(* CoDeSys 2.3 project: test.pro *)
(* Title: cy-wg-06 - ClevergyAS *)
(* Author: Andrea Ravasio *)
(* Libraries: Standard.lib 8.11.10 12:37:48, Util.lib 26.9.14 11:12:46, mod_com.lib 8.11.10 12:37:48, SerComm.lib 31.5.11 09:06:48, Serial_Interface_01.lib 22.4.13 12:50:14, 32_Bit\Modb_l05.lib 8.8.11 17:34:10, WagoLibIdent.lib 25.2.13 13:49:34, WagoLibStatus.lib 8.11.10 12:37:48, SysLibFile.lib 8.11.10 12:37:48, SysLibRtc.lib 8.11.10 12:37:48, SysLibSockets.lib 5.5.11 09:22:24, SysLibEvent.lib 8.11.10 12:37:48, SysLibPlcCtrl.lib 8.11.10 12:37:48, SysLibCallback.lib 8.11.10 12:37:48, Ethernet.lib 8.11.10 12:37:48, WagoLibModbus_IP_01.lib 26.5.15 11:20:08, WagoLibMBX_01.lib 20.3.12 16:32:38, LON_01.lib 28.9.12 14:05:10 *)

(* PLC configuration (modules and I/O channels)
0750-1506 8DI / 8DO 24V DC 0.5A [Type_34_8_Channels] node 0, in %IB32 out %QB8 {INTTypePAAssignment = PLC; INTTypeModule = plugged}
  VPN_ST1 AT %IX16.0 [BOOLOnX_I] Ch_1 Digital input
  LAMP_AL AT %QX4.0 [BOOLOnX_Q] Ch_1 Digital output
  KEY_QE_ST AT %IX16.1 [BOOLOnX_I] Ch_2 Digital input
  CIR05_EN AT %QX4.1 [BOOLOnX_Q] Ch_2 Digital output
  CIR06_AL AT %IX16.2 [BOOLOnX_I] Ch_3 Digital input
  CIR03_EN AT %QX4.2 [BOOLOnX_Q] Ch_3 Digital output
  CIR06_ST AT %IX16.3 [BOOLOnX_I] Ch_4 Digital input
  CIR04_EN AT %QX4.3 [BOOLOnX_Q] Ch_4 Digital output
  CIR06_AUT AT %IX16.4 [BOOLOnX_I] Ch_5 Digital input
  CIR02_EN AT %QX4.4 [BOOLOnX_Q] Ch_5 Digital output
  CIR05_AL AT %IX16.5 [BOOLOnX_I] Ch_6 Digital input
  CIR01_EN AT %QX4.5 [BOOLOnX_Q] Ch_6 Digital output
  CIR05_ST AT %IX16.6 [BOOLOnX_I] Ch_7 Digital input
  CAL01_Rst_Bruc AT %QX4.6 [BOOLOnX_Q] Ch_7 Digital output
  CIR05_AUT AT %IX16.7 [BOOLOnX_I] Ch_8 Digital input
  CAL01_On_Off AT %QX4.7 [BOOLOnX_Q] Ch_8 Digital output
0750-0430 8 DI 24 V DC 3.0ms [Type_1_8_Channels] node 1, in %IB32 out %QB8 {INTTypePAAssignment = PLC; INTTypeModule = plugged}
  CIR02_ST AT %IX16.8 [BOOLOnX_I] Ch_1 Digital input
  CIR01_AUT AT %IX16.9 [BOOLOnX_I] Ch_2 Digital input
  CIR03_AL AT %IX16.10 [BOOLOnX_I] Ch_3 Digital input
  CIR04_ST AT %IX16.11 [BOOLOnX_I] Ch_4 Digital input
  CIR04_AL AT %IX16.12 [BOOLOnX_I] Ch_5 Digital input
  CIR02_AL AT %IX16.13 [BOOLOnX_I] Ch_6 Digital input
  CIR01_ST AT %IX16.14 [BOOLOnX_I] Ch_7 Digital input
  CAL01_ST AT %IX16.15 [BOOLOnX_I] Ch_8 Digital input
0750-0430 8 DI 24 V DC 3.0ms [Type_1_8_Channels] node 2, in %IB33 out %QB9 {INTTypePAAssignment = PLC; INTTypeModule = plugged}
  CAL01_AL AT %IX17.0 [BOOLOnX_I] Ch_1 Digital input
  CIR03_AUT AT %IX17.1 [BOOLOnX_I] Ch_2 Digital input
  CTL01_ST AT %IX17.2 [BOOLOnX_I] Ch_3 Digital input
  CIR01_AL AT %IX17.3 [BOOLOnX_I] Ch_4 Digital input
  CIR02_AUT AT %IX17.4 [BOOLOnX_I] Ch_5 Digital input
  ALARM_PM_PB_TB AT %IX17.5 [BOOLOnX_I] Ch_6 Digital input
  CIR03_ST AT %IX17.6 [BOOLOnX_I] Ch_7 Digital input
  CIR04_AUT AT %IX17.7 [BOOLOnX_I] Ch_8 Digital input
0750-0504 4 DO 24V DC 0.5A [Type_10_4_Channels] node 3, in %IB34 out %QB9 {INTTypePAAssignment = PLC; INTTypeModule = plugged}
  CIR06_EN AT %QX4.8 [BOOLOnX_Q] Ch_1 Digital output
  AT %QX4.9 [BOOLOnX_Q] Ch_2 Digital output
  AT %QX4.10 [BOOLOnX_Q] Ch_3 Digital output
  AT %QX4.11 [BOOLOnX_Q] Ch_4 Digital output
0750-0464#04 2/4 AI RTD / ADJ./ HA [Type_44_4_Channels] node 5, in %IB32 out %QB4 {INTTypePAAssignment = PLC; INTTypeModule = plugged}
  AT %IW0 [INTOnW_I] Ch_1 signed Input value
  AT %IW1 [INTOnW_I] Ch_2 signed Input value
  AT %IW2 [INTOnW_I] Ch_3 signed Input value
  T_S04 AT %IW3 [INTOnW_I] Ch_4 signed Input value
0750-0464#04 2/4 AI RTD / ADJ./ HA [Type_44_4_Channels] node 6, in %IB32 out %QB4 {INTTypePAAssignment = PLC; INTTypeModule = plugged}
  T_S05 AT %IW4 [INTOnW_I] Ch_1 signed Input value
  T_S08 AT %IW5 [INTOnW_I] Ch_2 signed Input value
  T_S06 AT %IW6 [INTOnW_I] Ch_3 signed Input value
  T_S09 AT %IW7 [INTOnW_I] Ch_4 signed Input value
0750-0464#04 2/4 AI RTD / ADJ./ HA [Type_44_4_Channels] node 7, in %IB40 out %QB4 {INTTypePAAssignment = PLC; INTTypeModule = plugged}
  T_S12 AT %IW8 [INTOnW_I] Ch_1 signed Input value
  T_S14 AT %IW9 [INTOnW_I] Ch_2 signed Input value
  T_S13 AT %IW10 [INTOnW_I] Ch_3 signed Input value
  T_S11 AT %IW11 [INTOnW_I] Ch_4 signed Input value
0753-0653/0003-0000#03 RS485 Interface (Adjustable), 3 Bytes [Type_21_1_Channels] node 8, in %IB48 out %QB4 {INTTypePAAssignment = PLC; INTTypeModule = plugged}
  AT %IX12.0 [BOOLOnX_I] Transmission acknowledgement
  AT %IX12.1 [BOOLOnX_I] Reception request
  AT %IX12.2 [BOOLOnX_I] Initialization acknowledgement
  AT %IX12.3 [BOOLOnX_I] Input buffer is full
  AT %IX12.4 [BOOLOnX_I] Number of received characters Bit 0
  AT %IX12.5 [BOOLOnX_I] Number of received characters Bit 1
  AT %IX12.6 [BOOLOnX_I] Number of received characters Bit 2
  AT %IB25 [BYTEOnB_I] Input data Byte 0
  AT %IB26 [BYTEOnB_I] Input data Byte 1
  AT %IB27 [BYTEOnB_I] Input data Byte 2
  AT %QX0.0 [BOOLOnX_Q] Transmission request
  AT %QX0.1 [BOOLOnX_Q] Reception acknowledgement
  AT %QX0.2 [BOOLOnX_Q] Initialization request
  AT %QX0.4 [BOOLOnX_Q] Number of characters Bit 0
  AT %QX0.5 [BOOLOnX_Q] Number of characters Bit 1
  AT %QX0.6 [BOOLOnX_Q] Number of characters Bit 2
  AT %QB1 [BYTEOnB_Q] Output data Byte 0
  AT %QB2 [BYTEOnB_Q] Output data Byte 1
  AT %QB3 [BYTEOnB_Q] Output data Byte 2
0750-0478 2 AI 0-10V 16 Bit S.E. [Type_8_2_Channels] node 9, in %IB56 out %QB4 {INTTypePAAssignment = PLC; INTTypeModule = plugged}
  VRD02_ST AT %IW14 [WORDOnW_I] Ch_1 Input word
  VRD01_ST AT %IW15 [WORDOnW_I] Ch_2 Input word
0750-0556 2 AO ±10V [Type_14_2_Channels] node 10, in %IB60 out %QB8 {INTTypePAAssignment = PLC; INTTypeModule = plugged}
  VRD02_CTRL AT %QW2 [WORDOnW_Q] Ch_1 Analog output
  VRD01_CTRL AT %QW3 [WORDOnW_Q] Ch_2 Analog output
Fieldbus variables [FB_VARS] node 1, in %IB0 out %QB0
Flag variables [FLAG_VARS] node 2, in %IB0 out %QB0
Modbus-Master [MB_MASTER] node 3, in %IB0 out %QB0
*)

(* Global variable list: Global_Constants *)
VAR_GLOBAL CONSTANT

	Plant_NAME			: STRING :='cySN:13 cyVER: E09 Asilo Nido Comunale Albino ';
	Plant_SN			: DWORD  :=13;	(* S/N Impianto di telecontrollo *)
	Plant_SW_VER		: WORD   :=1;		(* Versione SW installata *)


	(* Colour defines *)
	COLOR_RED			: DWORD	:= 16#2020F0;
	COLOR_YELLOW		: DWORD	:= 16#20F0F0;
	COLOR_GREEN			: DWORD	:= 16#20F020;
	COLOR_LIGHT_GREEN	: DWORD := 16#006000;

	(* Parameters *)
	Plant_DefaultTAmb	: INT	:=100;		(* [.1°C] Temperatura ambiente di default in caso di rottura sonda *)
	Plant_MaxRunTAmb	: INT   :=210; 		(* [.1°C] Temperatura ambiente massima funzionamento impianto *)
	Plant_AntiFreezeTAmb: INT   :=-40;		(* [.1°C] Antifreeze temperature, start circulators *)
	Plant_VRD_TAlarm	: INT   :=850; 		(* [.1°C] Temperatura di allarme VRD, blocco *)
	Plant_VRD_TMax		: INT   :=800; 		(* [.1°C] Setpoint massimo per uscita VRD *)
	Plant_VRD_TDefault	: INT	:=300;		(* [.1°C] Temperatura di default in caso di errore climatica *)
	Plant_CirOffDelay	: TIME	:=T#30m;	(* (Def.T#15m) Ritardo spegnimento pompe per ricircolo caldaia *)
	Plant_CirOnDelay	: TIME	:=T#15m;
	Plant_MaxWaterLoss	: WORD  :=2;		(* [lt/h] Massima perdita del circuito *)

	(* Filesystem *)
	FilesPath  			: STRING :='S:\';

	(* TCP Logger *)
	Logger_SERVER		: STRING:='';
	Logger_IP			: STRING:='192.168.100.3';
	Logger_PORT			: WORD  :=80;
	Logger_GETSTART		: STRING:='GET /cygmsrv/hsgm.ashx?';
	Logger_GETEND		: STRING:='$R$N$R$N';
	Logger_CHECK		: STRING:='True';
	Logger_CRLF			: STRING:='$R$N';
	Logger_DataFile		: STRING:='S:\LOG.DAT';
	Logger_DataFileOld	: STRING:='S:\LOG.BCK';
	Logger_IndexFile	: STRING:='S:\LOG.IDX';
	Logger_ConnRetries	: BYTE:=5;
	Logger_RecoverMsgs	: BYTE:=25;

	(* TCP Remote *)
	Remote_PORT			: WORD  :=10;
	Remote_WELCOME		: STRING:='Connected$R$N';
	Remote_OK			: STRING:='OK$R$N';
	Remote_ERROR		: STRING:='ERROR$R$N';

	(* TCP Sockets *)
	MAX_SEND_TCP_SERVER					 : DWORD:=3000;(*60000*)
	MAX_RECEIVE_TCP_SERVER				 : DWORD:=3000;
	MAX_RECEIVE_TCP_SERVER_SOCKET	 	 : DWORD:=1500;
	MAX_SEND_TCP_CLIENT					 : DWORD:=3000;(*15000*)
	MAX_RECEIVE_TCP_CLIENT				 : DWORD:=1500;
	MAX_RECEIVE_TCP_CLIENT_SOCKET		 : DWORD:=1500;
	MAX_RECEIVE_UDP_SERVER				 : INT  :=1472;
	MAX_RECEIVE_UDP_CLIENT				 : INT  :=1472;
	CONNECT_WATCHDOG_TIME				 : TIME :=t#10s;

END_VAR




VAR_GLOBAL
(*	TestNodoInterogato: BYTE;
	NodoDaInterrogare: BYTE;
	InibiscoModbus: BOOL;
 *)

	NodoDaInterrogarePDC: BYTE;
	InibiscoModbusPDC: BOOL;

END_VAR

(* Global variable list: Global_Retain *)
VAR_GLOBAL RETAIN PERSISTENT
	Mode_Manual : BOOL := FALSE;

	CAL01_Clima : typ_Clima;
	PDC01_Clima : typ_Clima;
	VRD01_Clima : typ_Clima;
	VRD02_Clima : typ_Clima;

	Ctl01_Counter	:	DWORD;	(* Water counter *)


(* Impostazioni di imipanto *)

	DelayAllarmeTemperaturaNonRaggiunta: INT:=60;
	DeltaInterventoAllarmeTempeaturaNonRaggiuta: INT:=400;
	OffsetSetPointManuale: INT:=50;							(* Offset al Setpoint manuale per comensare lo scambiatore *)
	OffsetSetPointManuale2: INT:=50;						(* Offset al Setpoint manuale per comensare lo scambiatore Aggiuntivo *)
	BitAbilitaBoost: BOOL:=TRUE;						(* Abilitiazione Boost *)
	RifOffsetBoost:INT;									(* Offset al Setpoint della Caldaia per azione di Boost *)

	SogliaMinStartAntigelo: INT:=50;
	SogliaMinStopAntigelo: INT:=80;
	BitAbilitaAntigelo: BOOL:=TRUE;

END_VAR

(* Global variable list: Global_Variables *)
VAR_GLOBAL

	SYS    : typ_SYS;
	Logger : typ_Logger;


	Lamp	:	LAMP_AL_GENERALE;
	T_AMB	:	INT;		(* Environment temperature *)

	(* Sonde di temperature Esistenti *)
	T_S01: INT;
	T_S02: INT;
	T_S03: INT;

	TPV01  : obj_TPV	:= ( ID:=1 ); 							   (* T_S01 Esterna ---- Presi dal LON  *)
	TPV02  : obj_TPV	:= ( ID:=2 , IN_WMIN:=50 , IN_WMAX:=800 ); (* T_S02 - CAL01 - T_Send ---- Presi dal LON*)
	TPV03  : obj_TPV	:= ( ID:=3 , IN_WMIN:=50 , IN_WMAX:=800 ); (* T_S03 Temp. Mandata ---- Presi dal LON*)


	TPV04  : obj_TPV	:= ( ID:=4 , IN_WMIN:=50 , IN_WMAX:=800 ); (* T_S04 Temp Bollitore*)
	TPV05  : obj_TPV	:= ( ID:=5 , IN_WMIN:=50 , IN_WMAX:=800 ); (* T_S05 Temp Controllo CIR02 *)
	TPV06  : obj_TPV	:= ( ID:=6 , IN_WMIN:=50 , IN_WMAX:=800 ); (* T_S06 Temp Controllo CIR06*)
	TPV08  : obj_TPV	:= ( ID:=8 , IN_WMIN:=50 , IN_WMAX:=800 ); (* T_S08 Temp Collettore Mandata *)
	TPV09  : obj_TPV	:= ( ID:=9 , IN_WMIN:=50 , IN_WMAX:=800 ); (* T_S09 Temp Collettore Ritorno *)

	TPV11  : obj_TPV	:= ( ID:=11 , IN_WMIN:=50 , IN_WMAX:=800 ); (* T_S11 Temp Ritorno scambiatore Acqua calda Sanitaria*)
	TPV12  : obj_TPV	:= ( ID:=12 , IN_WMIN:=50 , IN_WMAX:=800 ); (* T_S12 Temp ritorno Acqua scambiatore ACS*)
	TPV13  : obj_TPV	:= ( ID:=13 , IN_WMIN:=50 , IN_WMAX:=800 ); (* T_S13 Temp mandata Acqua scambiatore ACS*)
	TPV14  : obj_TPV	:= ( ID:=14 , IN_WMIN:=50 , IN_WMAX:=800 ); (* T_S14 Temp Mandata Utenze Acqua Sanitaria*)
	TPV15  : obj_TPV	:= ( ID:=15 , IN_WMIN:=50 , IN_WMAX:=800 ); (* T_S15 Temp Acqua Bollintore Bassa presa da PDC *)


	(* Caldaia *)

(*	CAL01  : obj_CAL_Generica := ( ID:=1,Plant_CAL_TMax:=1000,Plant_CAL_TDefault:=600, 	(* sicurezze sul set point *)
									KP_PID:= 10,	(* Parametri regolazine PID *)
									TN_PID:= 0,
									TV_PID:= 0,
									BandaMortaPID:= 20); *)
	CAL01  :obj_CAL_MGK_2_WOCK := (ID:=1);

	(* Cronothermostat *)
	THER01	:	obj_CRONTER := (ID:=1,Local_MaxRunTAmb:=250,Histeresys:=10);	(* Crono per CIR02 Radiatori *)
	THER02	:	obj_CRONTER := (ID:=2,Local_MaxRunTAmb:=250,Histeresys:=10);	(* Crono per CIR06 Radiatori *)
	THER03	:	obj_CRONTER := (ID:=3,Local_MaxRunTAmb:=250,Histeresys:=10);	(* Crono per CIR05 circolatore ACS *)
	THER04	:	obj_CRONTER := (ID:=4,Local_MaxRunTAmb:=800,Histeresys:=50);	(* CronoTermostato  per CIR03 e CIR4 Boiller ACS *)
	THER05	:	obj_CRONTER := (ID:=5,Local_MaxRunTAmb:=800,Histeresys:=50);	(* CronoTermostato  per CIR03 e CIR4 Boiller ACS *)
	THER06	:	obj_CRONTER := (ID:=6,Local_MaxRunTAmb:=800,Histeresys:=50);	(* CronoTermostato Per Pompa di Calore *)

	THER250	:	obj_CRONTER := (ID:=250, Local_MaxRunTAmb:=250,Histeresys:=10);


	(* Water counter - 2 PULSES/LITER *)
	CTL01	:	obj_CTL	:= (ID:=1, Peso:=10);


	(* Pompe Ciroclatori Singoli  *)
(*	CIR01	:	obj_CIR := (ID:=1, CIR_AUTO:=TRUE, OnDelay:=T#1s, OffDelay:=T#1m); (* sempre in funzione insieme alla Caldaia serve per evitare condense sul ritorno *) *)
	CIR02	:	obj_CIR := (ID:=2, CIR_AUTO:=TRUE, OnDelay:=T#1m, OffDelay:=T#30m);
	CIR03	:	obj_CIR := (ID:=3, CIR_AUTO:=TRUE, OnDelay:=T#1m, OffDelay:=T#30m);
	CIR04	:	obj_CIR := (ID:=4, CIR_AUTO:=TRUE, OnDelay:=T#1m, OffDelay:=T#30m);
	CIR05	:	obj_CIR := (ID:=5, CIR_AUTO:=TRUE, OnDelay:=T#1m, OffDelay:=T#30m);
	CIR06	:	obj_CIR := (ID:=6, CIR_AUTO:=TRUE, OnDelay:=T#1m, OffDelay:=T#30m);

	(* Valvole motorizzate Analogiche  *)
	VRD01	:	obj_VRD_02:= (ID:=1, fFeedback:=TRUE, ReducedRange := FALSE,Local_VRD_TAlarm:=800);
	VRD02	:	obj_VRD_02:= (ID:=2, fFeedback:=TRUE, ReducedRange := FALSE,Local_VRD_TAlarm:=800);

	(* Pompa di Calore  *)
	PDC01	:obj_MODBUS_THAITY_ELECTA:= (ID:=1, Address:=1);



	(** Communication **)
	(* ModBus *)
	MODB01	:	obj_MODBUS		:= (ID:=1, COM:=2, BAUDRATE:=BAUD_9600 ,N_STOPBits:=1,RS485:=TRUE,MB_timeOut:=t#500ms);



	CronEd	: obj_CRON_EDITOR;
	(**** SIMULATION ONLY ****)
	(*...*)
END_VAR

(* Data type in LON/Enumerations *)
TYPE alarm_type_t :
(
	AL_HEADER := -13,
	AL_FOOTER := -12,
	AL_DEBUG := -11,
	AL_INFO := -10,
	AL_SYSTEM_INFO := -6,
	AL_VALUE_INVALID := -5,
	AL_CONSTANT := -4,
	AL_OFFLINE := -3,
	AL_UNKNOWN := -2,
	AL_NUL := -1,
	AL_NO_CONDITION := 0,
	AL_ALM_CONDITION := 1,
	AL_TOT_SVC_ALM_1 := 2,
	AL_TOT_SVC_ALM_2 := 3,
	AL_TOT_SVC_ALM_3 := 4,
	AL_LOW_LMT_CLR_1 := 5,
	AL_LOW_LMT_CLR_2 := 6,
	AL_HIGH_LMT_CLR_1 := 7,
	AL_HIGH_LMT_CLR_2 := 8,
	AL_LOW_LMT_ALM_1 := 9,
	AL_LOW_LMT_ALM_2 := 10,
	AL_HIGH_LMT_ALM_1 := 11,
	AL_HIGH_LMT_ALM_2 := 12,
	AL_FIR_ALM := 13,
	AL_FIR_PRE_ALM := 14,
	AL_FIR_TRBL := 15,
	AL_FIR_SUPV := 16,
	AL_FIR_TEST_ALM := 17,
	AL_FIR_TEST_PRE_ALM := 18,
	AL_FIR_ENVCOMP_MAX := 19,
	AL_FIR_MONITOR_COND := 20,
	AL_FIR_MAINT_ALERT := 21,
	AL_FATAL_ERROR := 30,
	AL_ERROR := 31,
	AL_WARNING := 32
);
END_TYPE

(* Data type in Logger *)
TYPE en_Logger_ErrLev :
(
	EL_Log			:=0,
	EL_Wrn			:=1,
	EL_Alarm		:=2,
	EL_AlarmStop	:=3
);
END_TYPE

(* Data type in Logger *)
TYPE en_Logger_Status :
(
	S_Logger_UNKNOWN := 0,
	S_Logger_IDLE,
	S_Logger_WAITCONN,
	S_Logger_WAITTX,
	S_Logger_WAITRESP,
	S_Logger_ERROR
);
END_TYPE

(* Data type *)
TYPE en_SYS_Objects :
(
	EO_SYS		:=0,  (* PLC *)
	EO_VPN		:=1,  (* VPN *)
	EO_DOOR		:=2,  (* Door & access control *)

	EO_CAL		:=10, (* Caldaia *)
	EO_CIR		:=11, (* Circolatore *)
	EO_CRON		:=12, (* Crono-termostato *)
	EO_VRD		:=13, (* Valvola miscelatore pannelli *)
	EO_CTL		:=14, (* Contalitri *)
	EO_CTB		:=15, (* Contabilizzatore *)
	EO_TPV		:=16, (* Temperature probes values *)
	EO_PPV		:=17, (* Pressure probes values *)
	EO_PBV		:=18, (* Over-Pressure Alarms *)
	EO_TBV		:=19, (* Over-Temperature Alarms *)
	EO_PMV		:=20, (* Under-Pressure Alarms *)
	EO_GRU		:=21, (* Gruppo termico *)
	EO_PDC		:=22, (* Pompa di calore *)
	EO_SOL		:=23, (* Pannello solare termico *)
	EO_ESOL		:=24, (* Pannello solare fotovoltaico *)
	EO_GAS		:=25, (* Contatore GAS *)
	EO_PORT		:=26, (* Misuratore di portata *)
	EO_FPV		:=27, (* Flow probes values *)
	EO_ANZ		:=28, (* Analizzatore di rete *)
	EO_SCA		:=29, (* Signal Control Alarms *)
	EO_LUX		:=30, (* Base Illumination point *)
	EO_LUXM		:=31, (* Metered Illumination point *)
	EO_PSG		:=32, (* Sensore di passaggio *)
	EO_HVAC		:=33, (* Heating, Ventilating and Air Conditioning *)
	EO_HYGRV	:=34, (* Relative Humidity sensors value *)
	EO_COOV		:=35, (* Carbon Dioxide CO2 sensors value *)
	EO_INV		:=36, (* Inverter *)
	EO_STR		:=37, (* Smart string box *)

	EO_CIRD		:=39, (* Double CIR *)
	EO_ACS		:=40, (* Hot domestic water *)
	EO_FRG		:=41, (* Frigo *)
	EO_THER		:=42, (* Thermostat *)
	EO_CIRM		:=43, (* Modbus CIR *)
	EO_CIRDM	:=44, (* Modbus double CIR *)

	EO_ZGW			:=200,  (* ZigBee - Gateway *)
	EO_ZRM			:=201,	(* ZigBee - Repeater *)
	EO_ZREL			:=202,	(* ZigBee - Actuator rele *)
	EO_ZTHL			:=203,	(* ZigBee - Temperature Sensor *)

	EO_ASGW			:=250,	(* ASi - Gateway *)
	EO_ASCBI		:=251,	(* ASi - Input Board, Ciabatta *)

	EO_LON			:=1000, (* Bus - LON *)
	EO_MODBUS		:=1001, (* Bus - MODBUS *)
	EO_MBUS			:=1002, (* Bus - M-BUS *)
	EO_MODBUS_TCP	:=1003, (* Bus - MODBUS TCP *)

	EO_GENERIC		:=9000, (* Generic dataset *)
	EO_EXPO			:=9001 (* EXPO dataset *)
);
END_TYPE

(* Data type *)
TYPE en_SYS_Status :
(
	S_UNKNOWN  := 0,
	S_STARTUP,
	S_INIT_RTC,
	S_INIT_VAR,
	S_AUTOTEST,
	S_RUNNING,
	S_SHUTDOWN,
	S_HALT
);
END_TYPE

(* Data type in LON/Enumerations *)
TYPE file_request_t :
(
	FR_NUL := -1,
	FR_OPEN_TO_SEND := 0,
	FR_OPEN_TO_RECEIVE := 1,
	FR_CLOSE_FILE := 2,
	FR_CLOSE_DELETE_FILE := 3,
	FR_DIRECTORY_LOOKUP := 4,
	FR_OPEN_TO_SEND_RA := 5,
	FR_OPEN_TO_RECEIVE_RA := 6
);
END_TYPE

(* Data type in LON/Enumerations *)
TYPE file_status_t :
(
	FS_NUL := -1,
	FS_XFER_OK := 0,
	FS_LOOKUP_OK := 1,
	FS_OPEN_FAIL := 2,
	FS_LOOKUP_ERR := 3,
	FS_XFER_UNDERWAY := 4,
	FS_IO_ERR := 5,
	FS_TIMEOUT_ERR := 6,
	FS_WINDOW_ERR := 7,
	FS_AUTH_ERR := 8,
	FS_ACCESS_UNAVAIL := 9,
	FS_SEEK_INVALID := 10,
	FS_SEEK_WAIT := 11
);
END_TYPE

(* Data type in LON/Enumerations *)
TYPE hvac_t :
(
	HVAC_NUL := -1,
	HVAC_AUTO := 0,
	HVAC_HEAT := 1,
	HVAC_MRNG_WRMUP := 2,
	HVAC_COOL := 3,
	HVAC_NIGHT_PURGE := 4,
	HVAC_PRE_COOL := 5,
	HVAC_OFF := 6,
	HVAC_TEST := 7,
	HVAC_EMERG_HEAT := 8,
	HVAC_FAN_ONLY := 9,
	HVAC_FREE_COOL := 10,
	HVAC_ICE := 11,
	HVAC_MAX_HEAT := 12,
	HVAC_ECONOMY := 13,
	HVAC_DEHUMID := 14,
	HVAC_CALIBRATE := 15,
	HVAC_EMERG_COOL := 16,
	HVAC_EMERG_STEAM := 17,
	HVAC_MAX_COOL := 18,
	HVAC_HVC_LOAD := 19,
	HVAC_NO_LOAD := 20
);
END_TYPE

(* Data type in LON/Enumerations *)
TYPE object_request_t :
(
	RQ_NUL := -1,
	RQ_NORMAL := 0,
	RQ_DISABLED := 1,
	RQ_UPDATE_STATUS := 2,
	RQ_SELF_TEST := 3,
	RQ_UPDATE_ALARM := 4,
	RQ_REPORT_MASK := 5,
	RQ_OVERRIDE := 6,
	RQ_ENABLE := 7,
	RQ_RMV_OVERRIDE := 8,
	RQ_CLEAR_STATUS := 9,
	RQ_CLEAR_ALARM := 10,
	RQ_ALARM_NOTIFY_ENABLED := 11,
	RQ_ALARM_NOTIFY_DISABLED := 12,
	RQ_MANUAL_CTRL := 13,
	RQ_REMOTE_CTRL := 14,
	RQ_PROGRAM := 15,
	RQ_CLEAR_RESET := 16,
	RQ_RESET := 17,
	RQ_CLEAR_LOG := 18,
	RQ_LOAD_PROGRAM := 19,
	RQ_RUN_PROGRAM := 20,
	RQ_HALT_PROGRAM := 21,
	RQ_RESTART_PROGRAM := 22,
	RQ_UNLOAD_PROGRAM := 23,
	RQ_STEP_PROGRAM := 24
);
END_TYPE

(* Data type in LON/Enumerations *)
TYPE priority_level_t :
(
	PR_NUL := -1,
	PR_LEVEL_0 := 0,
	PR_LEVEL_1 := 1,
	PR_LEVEL_2 := 2,
	PR_LEVEL_3 := 3,
	PR_1 := 4,
	PR_2 := 5,
	PR_3 := 6,
	PR_4 := 7,
	PR_6 := 8,
	PR_8 := 9,
	PR_10 := 10,
	PR_16 := 11
);
END_TYPE

(* Data type in Plant_Objects *)
TYPE typ_Clima : (* CURVA CLIMATICA *)
STRUCT
	InitOK:		BOOL;
	Points: 	ARRAY [0..10] OF POINT;
END_STRUCT
END_TYPE

(* Data type in Plant_Objects *)
TYPE typ_Cron_Calendar :
STRUCT
	Profile		: ARRAY[0..384] OF BYTE;
END_STRUCT
END_TYPE

(* Data type in Plant_Objects *)
TYPE typ_Cron_Jolly :
STRUCT
	Start		: DT;
	End			: DT;
	Temp		: WORD;
	Flags		: WORD; (* B0:Enabled B1..B15:Unused *)
END_STRUCT
END_TYPE

(* Data type in Plant_Objects *)
TYPE typ_Cron_Profile :
STRUCT
	Flags		: WORD;
	Setpoint	: ARRAY [0..95] OF WORD;
END_STRUCT
END_TYPE

(* Data type in Logger *)
TYPE typ_Logger :
STRUCT
	Status		: en_Logger_Status;

	SendReq		: BOOL;
	SendIdx		: DWORD;
	SendData	: ARRAY [0..MAX_SEND_TCP_CLIENT] OF BYTE;
	SendLen		: DINT;

	TData		: ARRAY [0..MAX_SEND_TCP_CLIENT] OF BYTE;
	TLen		: DINT;

	LastIdxPos	: DWORD;

	(* Temporary variables used by objects *)
	s1			: STRING(256);
	i1			: WORD;

END_STRUCT
END_TYPE

(* Data type in Plant_Objects *)
TYPE typ_MODBUS_ABB_DMTME72 :
STRUCT
	V_3P		: DWORD; (* V *)
	V_L1N		: DWORD;
	V_L2N		: DWORD;
	V_L3N		: DWORD;
	V_L1L2		: DWORD;
	V_L2L3		: DWORD;
	V_L3L1		: DWORD;
	I_3P		: DWORD; (* 10^-3 A *)
	I_L1		: DWORD;
	I_L2		: DWORD;
	I_L3		: DWORD;
	PF_3P		: DINT;	 (* 10^-3 *)
	PF_L1		: DINT;
	PF_L2		: DINT;
	PF_L3		: DINT;
	COS_3P		: DINT;  (*NO!*)
	COS_L1		: DINT;
	COS_L2		: DINT;
	COS_L3		: DINT;
	VA_3P		: DWORD; (* VA *)(*NO!*)
	VA_L1		: DWORD;
	VA_L2		: DWORD;
	VA_L3		: DWORD;
	P_3P		: DWORD; (* W *)
	P_L1		: DWORD;
	P_L2		: DWORD;
	P_L3		: DWORD;
	Q_3P		: DWORD; (* VAr *)
	Q_L1		: DWORD;
	Q_L2		: DWORD;
	Q_L3		: DWORD;

	WH_3P		: DWORD; (* 10^-1 kWh *)
	VARH_3P		: DWORD; (* 10^-1 kVArh *)
	FREQ		: DWORD; (* 10^-3 Hz *)

	I_L1_Max	: DWORD;
	I_L2_Max	: DWORD;
	I_L3_Max	: DWORD;
	P_3P_Max	: DWORD;
	Q_3P_Max	: DWORD;
	P_3P_Avg15m	: DWORD;

END_STRUCT
END_TYPE

(* Data type in Plant_Objects *)
TYPE typ_MODBUS_CIR :
STRUCT
	PumpStatus		:	WORD;
	PumpFault		:	BOOL;
	PumpBoardTemp	:	INT;	(* Electonic board temperature  [°C] *)
	PumpVoltage		:	WORD;	(* Input voltage rms [V] *)
	PumpCurrent		:	WORD;	(* Output current [E-3 A]	*)
	PumpRPM			:	WORD;	(* Round per minute [rpm] *)
	PumpPower		:	WORD;	(* Power [W] *)
	PumpOpTime		:	DWORD;	(* Pump operating time [h] *)
	PumpHead		:	WORD;	(* [E-1 m] *)
	PumpFlow		:	WORD;	(* Extimated flow [E-1 m3/h] *)
	PumpLiqTemp		:	WORD;	(* Liquid temperature [°C] *)
	PumpAlarm		:	ARRAY [0..14] OF WORD;

END_STRUCT
END_TYPE

(* Data type in Plant_Objects *)
TYPE typ_MODBUS_ELGAS_MINIELCOR :
STRUCT
	Vb			: ARRAY [0..3] OF WORD;	(* m^3 *)
	Vm			: DWORD;				(* m^3 *)
	P			: REAL;					(* bar *)
	T			: REAL;					(* °C *)
	C			: REAL;
	Vbs			: ARRAY [0..3] OF WORD;	(* m^3 *)
	Vb_d_d		: ARRAY [0..3] OF WORD;	(* m^3 *)
	Vb_d_m		: ARRAY [0..3] OF WORD;	(* m^3 *)
	Vm_d_d		: DWORD;				(* m^3 *)
	Q			: REAL;					(* m^3/h *)
	Qb			: REAL;					(* m^3/h *)

	BC_EVC		: REAL;			(* % *)
	BV_EVC		: REAL;			(* V *)
	D_Err		: WORD;			(* 0:OK, 1:FAIL *)
	Status		: DWORD;		(* Status bits *)

END_STRUCT
END_TYPE

(* Data type in Plant_Objects *)
TYPE typ_MODBUS_FRER_IQ96U2 :
STRUCT
	V_L1N		: DWORD; (* 10^-3 V *)
	V_L2N		: DWORD;
	V_L3N		: DWORD;
	V_L1L2		: DWORD;
	V_L2L3		: DWORD;
	V_L3L1		: DWORD;
	I_L1		: DWORD; (* 10^-3 I *)
	I_L2		: DWORD;
	I_L3		: DWORD;
	FREQ		: DWORD; (* 10^-3 Hz *)
	P_3P		: DWORD; (* W *)
	Q_3P		: DWORD; (* VAr *)
	PF_3P		: DINT;	 (* 10^-3 *)
	WH_3P		: DWORD; (* Wh *)
	VARH_3P		: DWORD; (* VArh *)
	MULT		: DWORD;

	WH_3P_NEG	: DWORD; (* Wh *)
	VARH_3P_NEG : DWORD; (* VArh *)
	S_3P		: DWORD; (* VA *)

	PF_L1		: DWORD; (* 10^-3 *)
	PF_L2		: DWORD; (* 10^-3 *)
	PF_L3		: DWORD; (* 10^-3 *)

	P_3P_Max	: DWORD;
	P_3P_Avg15m	: DWORD;
	I_L1_Max	: DWORD;
	I_L2_Max	: DWORD;
	I_L3_Max	: DWORD;
	I_L1_Avg15m	: DWORD;
	I_L2_Avg15m	: DWORD;
	I_L3_Avg15m	: DWORD;

END_STRUCT
END_TYPE

(* Data type in Plant_Objects *)
TYPE typ_MODBUS_VAR : (* Gestione parametri MODBUS *)
STRUCT
	SlaveAddress	: BYTE;
	FunCode			: BYTE;
	FunAddress		: WORD;
	Refresh_Time	: BYTE; (* 0:No refresh x:Refresh in seconds *)
	Refresh_Cnt		: BYTE; (* INTERNAL *)
	Variable		: POINTER TO WORD;
	Variable_Size	: BYTE;
	Variable_Mirror : WORD; (* INTERNAL [Force refresh on read variables when <>0] *)
END_STRUCT
END_TYPE

(* Data type *)
TYPE typ_SYS :
STRUCT
	Status			: en_SYS_Status;
	Warning			: BOOL;
	Alarm			: BOOL;
	AlarmStop		: BOOL;

	Time_LogString	: STRING;
	Time_Year		: WORD;
	Time_Month		: BYTE;
	Time_Day		: BYTE;
	Time_Hour		: BYTE;
	Time_Minute		: BYTE;

	Time_CT_DT		: DT;
	Time_CT_Day		: WORD;
	Time_CT_Quarter	: BYTE;

	LastLogs_Idx	: BYTE;
	LastLogs_Dat	: ARRAY[0..5] OF STRING;
	LastLogs_Msg	: ARRAY[0..5] OF STRING;

END_STRUCT
END_TYPE

(* Data type in Plant_Objects *)
TYPE typ_VisuStrutturaMbus :
STRUCT

	sdNodoPresente: STRING(16);
	sdEnergia: STRING(16);
	sdPotenza: STRING(16);
	sdVolume: STRING(16);
	sdFlow: STRING(16);
	sdTempIngresso: STRING(8);
	sdTempaUscita: STRING(8);
	sdTempDelta: STRING(8);

END_STRUCT
END_TYPE

(* Data type in LON/NetworkVariables *)
TYPE typSnvtAlarm : 
STRUCT
	abLocation : ARRAY[0..5] OF BYTE;
	wObjectId : WORD;
	bAlarmType : BYTE (* enum type alarm_type_t *);
	bPriorityLevel : BYTE (* enum type priority_level_t *);
	wIndexToSnvt : WORD;
	abValue : ARRAY[0..3] OF BYTE;
	wYear : WORD;
	bMonth : BYTE;
	bDay : BYTE;
	bHour : BYTE;
	bMinute : BYTE;
	bSecond : BYTE;
	wMillisecond : WORD;
	abAlarmLimit : ARRAY[0..3] OF BYTE;
	bStatusInformation : BYTE; (* bit allocation of bStatusInformation:
	bit 0: NVI update counter LSB
	bit 1: NVI update counter
	bit 2: NVI update counter
	bit 3: NVI update counter MSB
	bit 4: timeout for NVI occurs (MaxRcvTime expired)
	bit 5: reserved
	bit 6: reserved
	bit 7: force NVO update *)
	bInternalUseOnly : BYTE; (* Do not use this byte in your application! *)
END_STRUCT
END_TYPE

(* Data type in LON/NetworkVariables *)
TYPE typSnvtFilePos : 
STRUCT
	diRwPtr : DINT;
	wRwLength : WORD;
	bStatusInformation : BYTE; (* bit allocation of bStatusInformation:
	bit 0: NVI update counter LSB
	bit 1: NVI update counter
	bit 2: NVI update counter
	bit 3: NVI update counter MSB
	bit 4: timeout for NVI occurs (MaxRcvTime expired)
	bit 5: reserved
	bit 6: reserved
	bit 7: force NVO update *)
	bInternalUseOnly : BYTE; (* Do not use this byte in your application! *)
END_STRUCT
END_TYPE

(* Data type in LON/NetworkVariables *)
TYPE typSnvtFileReq : 
STRUCT
	bRequest : BYTE (* enum type file_request_t *);
	wIndex : WORD;
	wReceiveTimeout : WORD;
	abDestAddress : ARRAY[0..4] OF BYTE (* union declaration *);
	bAuthOn : BYTE;
	bPrioOn : BYTE;
	bStatusInformation : BYTE; (* bit allocation of bStatusInformation:
	bit 0: NVI update counter LSB
	bit 1: NVI update counter
	bit 2: NVI update counter
	bit 3: NVI update counter MSB
	bit 4: timeout for NVI occurs (MaxRcvTime expired)
	bit 5: reserved
	bit 6: reserved
	bit 7: force NVO update *)
	bInternalUseOnly : BYTE; (* Do not use this byte in your application! *)
END_STRUCT
END_TYPE

(* Data type in LON/NetworkVariables *)
TYPE typSnvtFileStatus : 
STRUCT
	bStatus : BYTE (* enum type file_status_t *);
	wNumberOfFiles : WORD;
	wSelectedFile : WORD;
	abAdr : ARRAY[0..21] OF BYTE (* union declaration *);
	bStatusInformation : BYTE; (* bit allocation of bStatusInformation:
	bit 0: NVI update counter LSB
	bit 1: NVI update counter
	bit 2: NVI update counter
	bit 3: NVI update counter MSB
	bit 4: timeout for NVI occurs (MaxRcvTime expired)
	bit 5: reserved
	bit 6: reserved
	bit 7: force NVO update *)
	bInternalUseOnly : BYTE; (* Do not use this byte in your application! *)
END_STRUCT
END_TYPE

(* Data type in LON/NetworkVariables *)
TYPE typSnvtHvacMode : 
STRUCT
	bSnvtHvacMode : BYTE (* enum type hvac_t *);
	bStatusInformation : BYTE; (* bit allocation of bStatusInformation:
	bit 0: NVI update counter LSB
	bit 1: NVI update counter
	bit 2: NVI update counter
	bit 3: NVI update counter MSB
	bit 4: timeout for NVI occurs (MaxRcvTime expired)
	bit 5: reserved
	bit 6: reserved
	bit 7: force NVO update *)
	bInternalUseOnly : BYTE; (* Do not use this byte in your application! *)
END_STRUCT
END_TYPE

(* Data type in LON/NetworkVariables *)
TYPE typSnvtObjRequest : 
STRUCT
	wObjectId : WORD;
	bObjectRequest : BYTE (* enum type object_request_t *);
	bStatusInformation : BYTE; (* bit allocation of bStatusInformation:
	bit 0: NVI update counter LSB
	bit 1: NVI update counter
	bit 2: NVI update counter
	bit 3: NVI update counter MSB
	bit 4: timeout for NVI occurs (MaxRcvTime expired)
	bit 5: reserved
	bit 6: reserved
	bit 7: force NVO update *)
	bInternalUseOnly : BYTE; (* Do not use this byte in your application! *)
END_STRUCT
END_TYPE

(* Data type in LON/NetworkVariables *)
TYPE typSnvtObjStatus : 
STRUCT
	wObjectId : WORD;
	bBitfieldByteOffset2 : BYTE (* bit field *);
	bBitfieldByteOffset3 : BYTE (* bit field *);
	bBitfieldByteOffset4 : BYTE (* bit field *);
	bBitfieldByteOffset5 : BYTE (* bit field *);
	bStatusInformation : BYTE; (* bit allocation of bStatusInformation:
	bit 0: NVI update counter LSB
	bit 1: NVI update counter
	bit 2: NVI update counter
	bit 3: NVI update counter MSB
	bit 4: timeout for NVI occurs (MaxRcvTime expired)
	bit 5: reserved
	bit 6: reserved
	bit 7: force NVO update *)
	bInternalUseOnly : BYTE; (* Do not use this byte in your application! *)
END_STRUCT
END_TYPE

(* Data type in LON/NetworkVariables *)
TYPE typSnvtState : 
STRUCT
	bBitfieldByteOffset0 : BYTE (* bit field *);
	bBitfieldByteOffset1 : BYTE (* bit field *);
	bStatusInformation : BYTE; (* bit allocation of bStatusInformation:
	bit 0: NVI update counter LSB
	bit 1: NVI update counter
	bit 2: NVI update counter
	bit 3: NVI update counter MSB
	bit 4: timeout for NVI occurs (MaxRcvTime expired)
	bit 5: reserved
	bit 6: reserved
	bit 7: force NVO update *)
	bInternalUseOnly : BYTE; (* Do not use this byte in your application! *)
END_STRUCT
END_TYPE

(* Data type in LON/NetworkVariables *)
TYPE typSnvtSwitch : 
STRUCT
	bValue : BYTE;
	siState : SINT;
	bStatusInformation : BYTE; (* bit allocation of bStatusInformation:
	bit 0: NVI update counter LSB
	bit 1: NVI update counter
	bit 2: NVI update counter
	bit 3: NVI update counter MSB
	bit 4: timeout for NVI occurs (MaxRcvTime expired)
	bit 5: reserved
	bit 6: reserved
	bit 7: force NVO update *)
	bInternalUseOnly : BYTE; (* Do not use this byte in your application! *)
END_STRUCT
END_TYPE

(* Data type in LON/NetworkVariables *)
TYPE typSnvtTemp : 
STRUCT
	wSnvtTemp : WORD;
	bStatusInformation : BYTE; (* bit allocation of bStatusInformation:
	bit 0: NVI update counter LSB
	bit 1: NVI update counter
	bit 2: NVI update counter
	bit 3: NVI update counter MSB
	bit 4: timeout for NVI occurs (MaxRcvTime expired)
	bit 5: reserved
	bit 6: reserved
	bit 7: force NVO update *)
	bInternalUseOnly : BYTE; (* Do not use this byte in your application! *)
END_STRUCT
END_TYPE

(* Data type in LON/NetworkVariables *)
TYPE typSnvtTempP : 
STRUCT
	iSnvtTempP : INT;
	bStatusInformation : BYTE; (* bit allocation of bStatusInformation:
	bit 0: NVI update counter LSB
	bit 1: NVI update counter
	bit 2: NVI update counter
	bit 3: NVI update counter MSB
	bit 4: timeout for NVI occurs (MaxRcvTime expired)
	bit 5: reserved
	bit 6: reserved
	bit 7: force NVO update *)
	bInternalUseOnly : BYTE; (* Do not use this byte in your application! *)
END_STRUCT
END_TYPE

(* Data type in LON/NetworkVariables *)
TYPE typSnvtTimeStamp : 
STRUCT
	iYear : INT;
	bMonth : BYTE;
	bDay : BYTE;
	bHour : BYTE;
	bMinute : BYTE;
	bSecond : BYTE;
	bStatusInformation : BYTE; (* bit allocation of bStatusInformation:
	bit 0: NVI update counter LSB
	bit 1: NVI update counter
	bit 2: NVI update counter
	bit 3: NVI update counter MSB
	bit 4: timeout for NVI occurs (MaxRcvTime expired)
	bit 5: reserved
	bit 6: reserved
	bit 7: force NVO update *)
	bInternalUseOnly : BYTE; (* Do not use this byte in your application! *)
END_STRUCT
END_TYPE

(* POU PLC_PRG, ST *)
PROGRAM PLC_PRG
VAR
	cont: INT;
END_VAR
cont:=Cont+1;
END_PROGRAM

(* Visualisation PLC_VISU
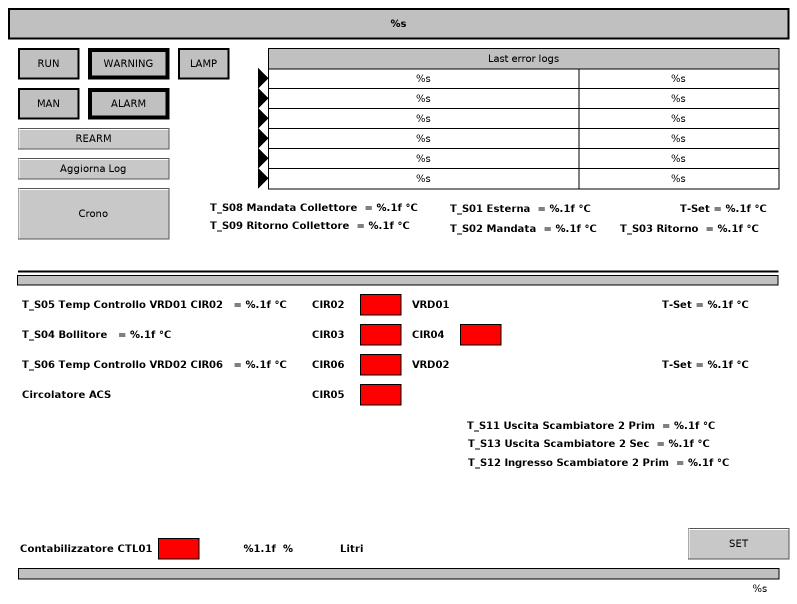
rectangle at (10,10)-(791,41): text "%s"; shows .Plant_NAME
rectangle at (530,580)-(771,601): text "%s"; shows Sys.Time_LogString
rounded rectangle at (20,50)-(81,81): text "RUN"; alarm colour if NOT Mode_Manual; runs INTERN ASSIGN Mode_Manual:=(FALSE)
rounded rectangle at (20,90)-(81,121): text "MAN"; alarm colour if Mode_Manual; runs INTERN ASSIGN Mode_Manual:=(TRUE)
rectangle at (580,70)-(781,91): text "%s"; shows Sys.LastLogs_Msg[0]
polygon at (260,170)-(270,190): invisible if Sys.LastLogs_Idx<>0
rectangle at (580,90)-(781,111): text "%s"; shows Sys.LastLogs_Msg[1]
polygon at (260,70)-(270,90): invisible if Sys.LastLogs_Idx<>1
rectangle at (580,110)-(781,131): text "%s"; shows Sys.LastLogs_Msg[2]
polygon at (260,90)-(270,110): invisible if Sys.LastLogs_Idx<>2
rectangle at (580,130)-(781,151): text "%s"; shows Sys.LastLogs_Msg[3]
polygon at (260,110)-(270,130): invisible if Sys.LastLogs_Idx<>3
rectangle at (580,150)-(781,171): text "%s"; shows Sys.LastLogs_Msg[4]
polygon at (260,130)-(270,150): invisible if Sys.LastLogs_Idx<>4
rectangle at (580,170)-(781,191): text "%s"; shows Sys.LastLogs_Msg[5]
polygon at (260,150)-(270,170): invisible if Sys.LastLogs_Idx<>5
rectangle at (270,70)-(581,91): text "%s"; shows Sys.LastLogs_Dat[0]
rectangle at (270,90)-(581,111): text "%s"; shows Sys.LastLogs_Dat[1]
rectangle at (270,110)-(581,131): text "%s"; shows Sys.LastLogs_Dat[2]
rectangle at (270,130)-(581,151): text "%s"; shows Sys.LastLogs_Dat[3]
rectangle at (270,150)-(581,171): text "%s"; shows Sys.LastLogs_Dat[4]
rectangle at (270,170)-(581,191): text "%s"; shows Sys.LastLogs_Dat[5]
rectangle at (90,90)-(171,121): text "ALARM"; alarm colour if Sys.Alarm; runs INTERN ASSIGN Mode_Manual:=(FALSE)
rectangle at (90,50)-(171,81): text "WARNING"; alarm colour if Sys.Warning; runs INTERN ASSIGN Mode_Manual:=(TRUE)
button at (20,130)-(171,151): text "REARM"; runs INTERN ASSIGN Sys.Alarm:=(FALSE);INTERN ASSIGN Sys.Warning:=(FALSE)
rectangle at (270,50)-(781,71): text "Last error logs"
rounded rectangle at (180,50)-(231,81): text "LAMP"; alarm colour if LAMP_AL
rectangle at (450,200)-(661,221): text "T_S01 Esterna  = %.1f °C"; shows INT_TO_REAL(.TPV01.AVG)/10
rectangle at (450,220)-(661,241): text "T_S02 Mandata  = %.1f °C"; shows INT_TO_REAL(.TPV02.AVG)/10
rectangle at (620,220)-(771,241): text "T_S03 Ritorno  = %.1f °C"; shows INT_TO_REAL(.TPV03.IN)/10
rectangle at (22,326)-(233,347): text "T_S04 Bollitore   = %.1f °C"; shows INT_TO_REAL(.TPV04.IN)/10
rectangle at (22,296)-(313,317): text "T_S05 Temp Controllo VRD01 CIR02   = %.1f °C"; shows INT_TO_REAL(.TPV05.IN)/10
rectangle at (22,356)-(303,377): text "T_S06 Temp Controllo VRD02 CIR06   = %.1f °C"; shows INT_TO_REAL(.TPV06.IN)/10
button at (20,160)-(171,181): text "Aggiorna Log"; taps PLC_PRG.HMI_AggiornaLog
button at (20,190)-(171,241): text "Crono"; opens VIS_CHONOEDITOR
rectangle at (680,200)-(781,221): text "T-Set = %.1f °C"; shows INT_TO_REAL(.CAL01.SetPointCaldaia)/10
rectangle at (312,296)-(363,317): text "CIR02"
rectangle at (412,296)-(463,317): text "VRD01"
rectangle at (312,326)-(363,347): text "CIR03"
rectangle at (412,326)-(463,347): text "CIR04"
rectangle at (312,386)-(363,407): text "CIR05"
rectangle at (312,356)-(363,377): text "CIR06"
rectangle at (412,356)-(463,377): text "VRD02"
rectangle at (20,540)-(181,561): text "Contabilizzatore CTL01"; shows INT_TO_REAL(.TPV06.IN)/10)
rectangle at (160,540)-(201,561): alarm colour if .CTL01.CTL_ST
rectangle at (210,540)-(331,561): text "%1.1f  %"; shows DINT_TO_REAL(.CTL01.COUNT)/10
button at (690,530)-(791,561): text "SET"; opens VIS_SET
rectangle at (340,540)-(381,561): text "Litri"; shows INT_TO_REAL(.TPV06.IN)/10)
rectangle at (362,296)-(403,317): alarm colour if .CIR02_ST
rectangle at (362,326)-(403,347): alarm colour if .CIR03_ST
rectangle at (362,356)-(403,377): alarm colour if .CIR06_ST
rectangle at (462,326)-(503,347): alarm colour if .CIR04_ST
rectangle at (362,386)-(403,407): alarm colour if .CIR05_ST
rectangle at (22,386)-(303,407): text "Circolatore ACS"; shows INT_TO_REAL(.TPV06.IN)/10
rectangle at (662,296)-(763,317): text "T-Set = %.1f °C"; shows INT_TO_REAL(.VRD01.Ctrl_SetPoint)/10
rectangle at (662,356)-(763,377): text "T-Set = %.1f °C"; shows INT_TO_REAL(.VRD02.Ctrl_SetPoint)/10
rectangle at (210,199)-(430,220): text "T_S08 Mandata Collettore  = %.1f °C"; shows INT_TO_REAL(.TPV08.AVG)/10
rectangle at (210,217)-(421,238): text "T_S09 Ritorno Collettore  = %.1f °C"; shows INT_TO_REAL(.TPV09.AVG)/10
rectangle at (467,417)-(733,438): text "T_S11 Uscita Scambiatore 2 Prim  = %.1f °C"; shows INT_TO_REAL(.TPV11.AVG)/10
rectangle at (468,435)-(759,456): text "T_S13 Uscita Scambiatore 2 Sec  = %.1f °C"; shows INT_TO_REAL(.TPV13.AVG)/10
rectangle at (468,454)-(759,475): text "T_S12 Ingresso Scambiatore 2 Prim  = %.1f °C"; shows INT_TO_REAL(.TPV12.AVG)/10
3 more shapes without text or variables
4 elements of other kinds (tables, trends, ...) not read
*)

(* Visualisation VIS_CHONOEDITOR
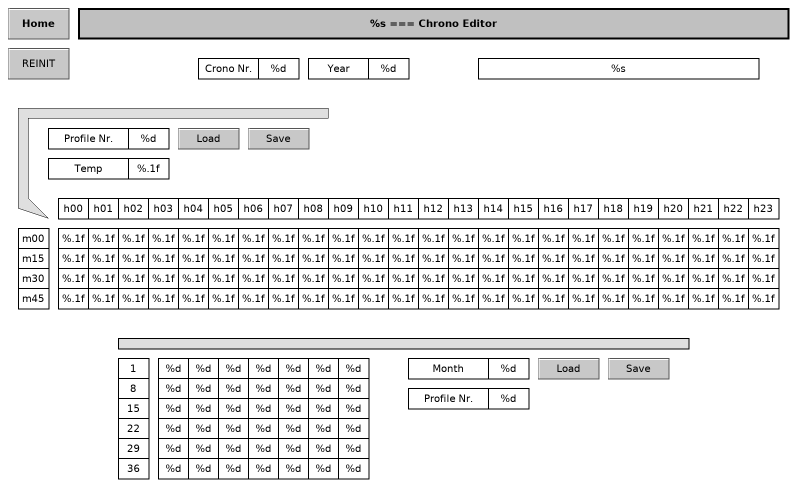
rectangle at (200,60)-(261,81): text "Crono Nr."
rectangle at (260,60)-(301,81): text "%d"; shows CronEd.CN_Sel; alarm colour if CronEd.CN_Sel<>CronEd.CN_Act; editable 1..6
rectangle at (50,130)-(131,151): text "Profile Nr."
rectangle at (130,130)-(171,151): text "%d"; shows CronEd.PR_Sel; alarm colour if CronEd.PR_Sel<>CronEd.PR_Act; editable 1..10
rectangle at (50,160)-(131,181): text "Temp"
rectangle at (130,160)-(171,181): text "%.1f"; shows CronEd.PR_TT; editable
button at (180,130)-(241,151): text "Load"; toggles CronEd.PR_Load
button at (250,130)-(311,151): text "Save"; toggles CronEd.PR_Save
rectangle at (20,230)-(51,251): text "m00"
rectangle at (20,250)-(51,271): text "m15"
rectangle at (20,270)-(51,291): text "m30"
rectangle at (20,290)-(51,311): text "m45"
rectangle at (80,10)-(791,41): text "%s === Chrono Editor"; shows .Plant_NAME
button at (10,10)-(71,41): text "Home"; opens PLC_VISU
rounded rectangle at (60,230)-(91,251): text "%.1f"; shows WORD_TO_REAL(CronEd.PR.Setpoint[0])/10; runs INTERN ASSIGN CronEd.PR.Setpoint[0]:=(REAL_TO_WORD(CronEd.PR_TT*10))
rounded rectangle at (60,250)-(91,271): text "%.1f"; shows WORD_TO_REAL(CronEd.PR.Setpoint[1])/10; runs INTERN ASSIGN CronEd.PR.Setpoint[1]:=(REAL_TO_WORD(CronEd.PR_TT*10))
rounded rectangle at (60,270)-(91,291): text "%.1f"; shows WORD_TO_REAL(CronEd.PR.Setpoint[2])/10; runs INTERN ASSIGN CronEd.PR.Setpoint[2]:=(REAL_TO_WORD(CronEd.PR_TT*10))
rounded rectangle at (60,290)-(91,311): text "%.1f"; shows WORD_TO_REAL(CronEd.PR.Setpoint[3])/10; runs INTERN ASSIGN CronEd.PR.Setpoint[3]:=(REAL_TO_WORD(CronEd.PR_TT*10))
rectangle at (60,200)-(91,221): text "h00"; runs INTERN ASSIGN CronEd.PR.Setpoint[0]:=(REAL_TO_WORD(CronEd.PR_TT*10));INTERN ASSIGN CronEd.PR.Setpoint[1]:=(REAL_TO_WORD(CronEd.PR_TT*10));INTERN ASSIGN CronEd.PR.Setpoint[2]:=(REAL_TO_WORD(CronEd.PR_TT*10));INTERN ASSIGN CronEd.PR.Setpoint[3]:=(REAL_TO_WORD(CronEd.PR_TT*10))
rounded rectangle at (90,230)-(121,251): text "%.1f"; shows WORD_TO_REAL(CronEd.PR.Setpoint[4])/10; runs INTERN ASSIGN CronEd.PR.Setpoint[4]:=(REAL_TO_WORD(CronEd.PR_TT*10))
rounded rectangle at (90,250)-(121,271): text "%.1f"; shows WORD_TO_REAL(CronEd.PR.Setpoint[5])/10; runs INTERN ASSIGN CronEd.PR.Setpoint[5]:=(REAL_TO_WORD(CronEd.PR_TT*10))
rounded rectangle at (90,270)-(121,291): text "%.1f"; shows WORD_TO_REAL(CronEd.PR.Setpoint[6])/10; runs INTERN ASSIGN CronEd.PR.Setpoint[6]:=(REAL_TO_WORD(CronEd.PR_TT*10))
rounded rectangle at (90,290)-(121,311): text "%.1f"; shows WORD_TO_REAL(CronEd.PR.Setpoint[7])/10; runs INTERN ASSIGN CronEd.PR.Setpoint[7]:=(REAL_TO_WORD(CronEd.PR_TT*10))
rectangle at (90,200)-(121,221): text "h01"; runs INTERN ASSIGN CronEd.PR.Setpoint[4]:=(REAL_TO_WORD(CronEd.PR_TT*10));INTERN ASSIGN CronEd.PR.Setpoint[5]:=(REAL_TO_WORD(CronEd.PR_TT*10));INTERN ASSIGN CronEd.PR.Setpoint[6]:=(REAL_TO_WORD(CronEd.PR_TT*10));INTERN ASSIGN CronEd.PR.Setpoint[7]:=(REAL_TO_WORD(CronEd.PR_TT*10))
rounded rectangle at (120,230)-(151,251): text "%.1f"; shows WORD_TO_REAL(CronEd.PR.Setpoint[8])/10; runs INTERN ASSIGN CronEd.PR.Setpoint[8]:=(REAL_TO_WORD(CronEd.PR_TT*10))
rounded rectangle at (120,250)-(151,271): text "%.1f"; shows WORD_TO_REAL(CronEd.PR.Setpoint[9])/10; runs INTERN ASSIGN CronEd.PR.Setpoint[9]:=(REAL_TO_WORD(CronEd.PR_TT*10))
rounded rectangle at (120,270)-(151,291): text "%.1f"; shows WORD_TO_REAL(CronEd.PR.Setpoint[10])/10; runs INTERN ASSIGN CronEd.PR.Setpoint[10]:=(REAL_TO_WORD(CronEd.PR_TT*10))
rounded rectangle at (120,290)-(151,311): text "%.1f"; shows WORD_TO_REAL(CronEd.PR.Setpoint[11])/10; runs INTERN ASSIGN CronEd.PR.Setpoint[11]:=(REAL_TO_WORD(CronEd.PR_TT*10))
rectangle at (120,200)-(151,221): text "h02"; runs INTERN ASSIGN CronEd.PR.Setpoint[8]:=(REAL_TO_WORD(CronEd.PR_TT*10));INTERN ASSIGN CronEd.PR.Setpoint[9]:=(REAL_TO_WORD(CronEd.PR_TT*10));INTERN ASSIGN CronEd.PR.Setpoint[10]:=(REAL_TO_WORD(CronEd.PR_TT*10));INTERN ASSIGN CronEd.PR.Setpoint[11]:=(REAL_TO_WORD(CronEd.PR_TT*10))
rounded rectangle at (150,230)-(181,251): text "%.1f"; shows WORD_TO_REAL(CronEd.PR.Setpoint[12])/10; runs INTERN ASSIGN CronEd.PR.Setpoint[12]:=(REAL_TO_WORD(CronEd.PR_TT*10))
rounded rectangle at (150,250)-(181,271): text "%.1f"; shows WORD_TO_REAL(CronEd.PR.Setpoint[13])/10; runs INTERN ASSIGN CronEd.PR.Setpoint[13]:=(REAL_TO_WORD(CronEd.PR_TT*10))
rounded rectangle at (150,270)-(181,291): text "%.1f"; shows WORD_TO_REAL(CronEd.PR.Setpoint[14])/10; runs INTERN ASSIGN CronEd.PR.Setpoint[14]:=(REAL_TO_WORD(CronEd.PR_TT*10))
rounded rectangle at (150,290)-(181,311): text "%.1f"; shows WORD_TO_REAL(CronEd.PR.Setpoint[15])/10; runs INTERN ASSIGN CronEd.PR.Setpoint[15]:=(REAL_TO_WORD(CronEd.PR_TT*10))
rectangle at (150,200)-(181,221): text "h03"; runs INTERN ASSIGN CronEd.PR.Setpoint[15]:=(REAL_TO_WORD(CronEd.PR_TT*10));INTERN ASSIGN CronEd.PR.Setpoint[14]:=(REAL_TO_WORD(CronEd.PR_TT*10));INTERN ASSIGN CronEd.PR.Setpoint[13]:=(REAL_TO_WORD(CronEd.PR_TT*10));INTERN ASSIGN CronEd.PR.Setpoint[12]:=(REAL_TO_WORD(CronEd.PR_TT*10))
rounded rectangle at (180,230)-(211,251): text "%.1f"; shows WORD_TO_REAL(CronEd.PR.Setpoint[16])/10; runs INTERN ASSIGN CronEd.PR.Setpoint[16]:=(REAL_TO_WORD(CronEd.PR_TT*10))
rounded rectangle at (180,250)-(211,271): text "%.1f"; shows WORD_TO_REAL(CronEd.PR.Setpoint[17])/10; runs INTERN ASSIGN CronEd.PR.Setpoint[17]:=(REAL_TO_WORD(CronEd.PR_TT*10))
rounded rectangle at (180,270)-(211,291): text "%.1f"; shows WORD_TO_REAL(CronEd.PR.Setpoint[18])/10; runs INTERN ASSIGN CronEd.PR.Setpoint[18]:=(REAL_TO_WORD(CronEd.PR_TT*10))
rounded rectangle at (180,290)-(211,311): text "%.1f"; shows WORD_TO_REAL(CronEd.PR.Setpoint[19])/10; runs INTERN ASSIGN CronEd.PR.Setpoint[19]:=(REAL_TO_WORD(CronEd.PR_TT*10))
rectangle at (180,200)-(211,221): text "h04"; runs INTERN ASSIGN CronEd.PR.Setpoint[19]:=(REAL_TO_WORD(CronEd.PR_TT*10));INTERN ASSIGN CronEd.PR.Setpoint[18]:=(REAL_TO_WORD(CronEd.PR_TT*10));INTERN ASSIGN CronEd.PR.Setpoint[17]:=(REAL_TO_WORD(CronEd.PR_TT*10));INTERN ASSIGN CronEd.PR.Setpoint[16]:=(REAL_TO_WORD(CronEd.PR_TT*10))
rounded rectangle at (210,230)-(241,251): text "%.1f"; shows WORD_TO_REAL(CronEd.PR.Setpoint[20])/10; runs INTERN ASSIGN CronEd.PR.Setpoint[20]:=(REAL_TO_WORD(CronEd.PR_TT*10))
rounded rectangle at (210,250)-(241,271): text "%.1f"; shows WORD_TO_REAL(CronEd.PR.Setpoint[21])/10; runs INTERN ASSIGN CronEd.PR.Setpoint[21]:=(REAL_TO_WORD(CronEd.PR_TT*10))
rounded rectangle at (210,270)-(241,291): text "%.1f"; shows WORD_TO_REAL(CronEd.PR.Setpoint[22])/10; runs INTERN ASSIGN CronEd.PR.Setpoint[22]:=(REAL_TO_WORD(CronEd.PR_TT*10))
rounded rectangle at (210,290)-(241,311): text "%.1f"; shows WORD_TO_REAL(CronEd.PR.Setpoint[23])/10; runs INTERN ASSIGN CronEd.PR.Setpoint[23]:=(REAL_TO_WORD(CronEd.PR_TT*10))
rectangle at (210,200)-(241,221): text "h05"; runs INTERN ASSIGN CronEd.PR.Setpoint[23]:=(REAL_TO_WORD(CronEd.PR_TT*10));INTERN ASSIGN CronEd.PR.Setpoint[22]:=(REAL_TO_WORD(CronEd.PR_TT*10));INTERN ASSIGN CronEd.PR.Setpoint[21]:=(REAL_TO_WORD(CronEd.PR_TT*10));INTERN ASSIGN CronEd.PR.Setpoint[20]:=(REAL_TO_WORD(CronEd.PR_TT*10))
rounded rectangle at (240,230)-(271,251): text "%.1f"; shows WORD_TO_REAL(CronEd.PR.Setpoint[24])/10; runs INTERN ASSIGN CronEd.PR.Setpoint[24]:=(REAL_TO_WORD(CronEd.PR_TT*10))
rounded rectangle at (240,250)-(271,271): text "%.1f"; shows WORD_TO_REAL(CronEd.PR.Setpoint[25])/10; runs INTERN ASSIGN CronEd.PR.Setpoint[25]:=(REAL_TO_WORD(CronEd.PR_TT*10))
rounded rectangle at (240,270)-(271,291): text "%.1f"; shows WORD_TO_REAL(CronEd.PR.Setpoint[26])/10; runs INTERN ASSIGN CronEd.PR.Setpoint[26]:=(REAL_TO_WORD(CronEd.PR_TT*10))
rounded rectangle at (240,290)-(271,311): text "%.1f"; shows WORD_TO_REAL(CronEd.PR.Setpoint[27])/10; runs INTERN ASSIGN CronEd.PR.Setpoint[27]:=(REAL_TO_WORD(CronEd.PR_TT*10))
rectangle at (240,200)-(271,221): text "h06"; runs INTERN ASSIGN CronEd.PR.Setpoint[27]:=(REAL_TO_WORD(CronEd.PR_TT*10));INTERN ASSIGN CronEd.PR.Setpoint[26]:=(REAL_TO_WORD(CronEd.PR_TT*10));INTERN ASSIGN CronEd.PR.Setpoint[25]:=(REAL_TO_WORD(CronEd.PR_TT*10));INTERN ASSIGN CronEd.PR.Setpoint[24]:=(REAL_TO_WORD(CronEd.PR_TT*10))
rounded rectangle at (270,230)-(301,251): text "%.1f"; shows WORD_TO_REAL(CronEd.PR.Setpoint[28])/10; runs INTERN ASSIGN CronEd.PR.Setpoint[28]:=(REAL_TO_WORD(CronEd.PR_TT*10))
rounded rectangle at (270,250)-(301,271): text "%.1f"; shows WORD_TO_REAL(CronEd.PR.Setpoint[29])/10; runs INTERN ASSIGN CronEd.PR.Setpoint[29]:=(REAL_TO_WORD(CronEd.PR_TT*10))
rounded rectangle at (270,270)-(301,291): text "%.1f"; shows WORD_TO_REAL(CronEd.PR.Setpoint[30])/10; runs INTERN ASSIGN CronEd.PR.Setpoint[30]:=(REAL_TO_WORD(CronEd.PR_TT*10))
rounded rectangle at (270,290)-(301,311): text "%.1f"; shows WORD_TO_REAL(CronEd.PR.Setpoint[31])/10; runs INTERN ASSIGN CronEd.PR.Setpoint[31]:=(REAL_TO_WORD(CronEd.PR_TT*10))
rectangle at (270,200)-(301,221): text "h07"; runs INTERN ASSIGN CronEd.PR.Setpoint[31]:=(REAL_TO_WORD(CronEd.PR_TT*10));INTERN ASSIGN CronEd.PR.Setpoint[30]:=(REAL_TO_WORD(CronEd.PR_TT*10));INTERN ASSIGN CronEd.PR.Setpoint[29]:=(REAL_TO_WORD(CronEd.PR_TT*10));INTERN ASSIGN CronEd.PR.Setpoint[28]:=(REAL_TO_WORD(CronEd.PR_TT*10))
rounded rectangle at (300,230)-(331,251): text "%.1f"; shows WORD_TO_REAL(CronEd.PR.Setpoint[32])/10; runs INTERN ASSIGN CronEd.PR.Setpoint[32]:=(REAL_TO_WORD(CronEd.PR_TT*10))
rounded rectangle at (300,250)-(331,271): text "%.1f"; shows WORD_TO_REAL(CronEd.PR.Setpoint[33])/10; runs INTERN ASSIGN CronEd.PR.Setpoint[33]:=(REAL_TO_WORD(CronEd.PR_TT*10))
rounded rectangle at (300,270)-(331,291): text "%.1f"; shows WORD_TO_REAL(CronEd.PR.Setpoint[34])/10; runs INTERN ASSIGN CronEd.PR.Setpoint[34]:=(REAL_TO_WORD(CronEd.PR_TT*10))
rounded rectangle at (300,290)-(331,311): text "%.1f"; shows WORD_TO_REAL(CronEd.PR.Setpoint[35])/10; runs INTERN ASSIGN CronEd.PR.Setpoint[35]:=(REAL_TO_WORD(CronEd.PR_TT*10))
rectangle at (300,200)-(331,221): text "h08"; runs INTERN ASSIGN CronEd.PR.Setpoint[35]:=(REAL_TO_WORD(CronEd.PR_TT*10));INTERN ASSIGN CronEd.PR.Setpoint[34]:=(REAL_TO_WORD(CronEd.PR_TT*10));INTERN ASSIGN CronEd.PR.Setpoint[33]:=(REAL_TO_WORD(CronEd.PR_TT*10));INTERN ASSIGN CronEd.PR.Setpoint[32]:=(REAL_TO_WORD(CronEd.PR_TT*10))
rounded rectangle at (330,230)-(361,251): text "%.1f"; shows WORD_TO_REAL(CronEd.PR.Setpoint[36])/10; runs INTERN ASSIGN CronEd.PR.Setpoint[36]:=(REAL_TO_WORD(CronEd.PR_TT*10))
rounded rectangle at (330,250)-(361,271): text "%.1f"; shows WORD_TO_REAL(CronEd.PR.Setpoint[37])/10; runs INTERN ASSIGN CronEd.PR.Setpoint[37]:=(REAL_TO_WORD(CronEd.PR_TT*10))
rounded rectangle at (330,270)-(361,291): text "%.1f"; shows WORD_TO_REAL(CronEd.PR.Setpoint[38])/10; runs INTERN ASSIGN CronEd.PR.Setpoint[38]:=(REAL_TO_WORD(CronEd.PR_TT*10))
rounded rectangle at (330,290)-(361,311): text "%.1f"; shows WORD_TO_REAL(CronEd.PR.Setpoint[39])/10; runs INTERN ASSIGN CronEd.PR.Setpoint[39]:=(REAL_TO_WORD(CronEd.PR_TT*10))
rectangle at (330,200)-(361,221): text "h09"; runs INTERN ASSIGN CronEd.PR.Setpoint[39]:=(REAL_TO_WORD(CronEd.PR_TT*10));INTERN ASSIGN CronEd.PR.Setpoint[38]:=(REAL_TO_WORD(CronEd.PR_TT*10));INTERN ASSIGN CronEd.PR.Setpoint[37]:=(REAL_TO_WORD(CronEd.PR_TT*10));INTERN ASSIGN CronEd.PR.Setpoint[36]:=(REAL_TO_WORD(CronEd.PR_TT*10))
rounded rectangle at (360,230)-(391,251): text "%.1f"; shows WORD_TO_REAL(CronEd.PR.Setpoint[40])/10; runs INTERN ASSIGN CronEd.PR.Setpoint[40]:=(REAL_TO_WORD(CronEd.PR_TT*10))
rounded rectangle at (360,250)-(391,271): text "%.1f"; shows WORD_TO_REAL(CronEd.PR.Setpoint[41])/10; runs INTERN ASSIGN CronEd.PR.Setpoint[41]:=(REAL_TO_WORD(CronEd.PR_TT*10))
rounded rectangle at (360,270)-(391,291): text "%.1f"; shows WORD_TO_REAL(CronEd.PR.Setpoint[42])/10; runs INTERN ASSIGN CronEd.PR.Setpoint[42]:=(REAL_TO_WORD(CronEd.PR_TT*10))
rounded rectangle at (360,290)-(391,311): text "%.1f"; shows WORD_TO_REAL(CronEd.PR.Setpoint[43])/10; runs INTERN ASSIGN CronEd.PR.Setpoint[43]:=(REAL_TO_WORD(CronEd.PR_TT*10))
rectangle at (360,200)-(391,221): text "h10"; runs INTERN ASSIGN CronEd.PR.Setpoint[43]:=(REAL_TO_WORD(CronEd.PR_TT*10));INTERN ASSIGN CronEd.PR.Setpoint[42]:=(REAL_TO_WORD(CronEd.PR_TT*10));INTERN ASSIGN CronEd.PR.Setpoint[41]:=(REAL_TO_WORD(CronEd.PR_TT*10));INTERN ASSIGN CronEd.PR.Setpoint[40]:=(REAL_TO_WORD(CronEd.PR_TT*10))
rounded rectangle at (390,230)-(421,251): text "%.1f"; shows WORD_TO_REAL(CronEd.PR.Setpoint[44])/10; runs INTERN ASSIGN CronEd.PR.Setpoint[44]:=(REAL_TO_WORD(CronEd.PR_TT*10))
rounded rectangle at (390,250)-(421,271): text "%.1f"; shows WORD_TO_REAL(CronEd.PR.Setpoint[45])/10; runs INTERN ASSIGN CronEd.PR.Setpoint[45]:=(REAL_TO_WORD(CronEd.PR_TT*10))
rounded rectangle at (390,270)-(421,291): text "%.1f"; shows WORD_TO_REAL(CronEd.PR.Setpoint[46])/10; runs INTERN ASSIGN CronEd.PR.Setpoint[46]:=(REAL_TO_WORD(CronEd.PR_TT*10))
rounded rectangle at (390,290)-(421,311): text "%.1f"; shows WORD_TO_REAL(CronEd.PR.Setpoint[47])/10; runs INTERN ASSIGN CronEd.PR.Setpoint[47]:=(REAL_TO_WORD(CronEd.PR_TT*10))
rectangle at (390,200)-(421,221): text "h11"; runs INTERN ASSIGN CronEd.PR.Setpoint[47]:=(REAL_TO_WORD(CronEd.PR_TT*10));INTERN ASSIGN CronEd.PR.Setpoint[46]:=(REAL_TO_WORD(CronEd.PR_TT*10));INTERN ASSIGN CronEd.PR.Setpoint[45]:=(REAL_TO_WORD(CronEd.PR_TT*10));INTERN ASSIGN CronEd.PR.Setpoint[44]:=(REAL_TO_WORD(CronEd.PR_TT*10))
rounded rectangle at (420,230)-(451,251): text "%.1f"; shows WORD_TO_REAL(CronEd.PR.Setpoint[48])/10; runs INTERN ASSIGN CronEd.PR.Setpoint[48]:=(REAL_TO_WORD(CronEd.PR_TT*10))
rounded rectangle at (420,250)-(451,271): text "%.1f"; shows WORD_TO_REAL(CronEd.PR.Setpoint[49])/10; runs INTERN ASSIGN CronEd.PR.Setpoint[49]:=(REAL_TO_WORD(CronEd.PR_TT*10))
rounded rectangle at (420,270)-(451,291): text "%.1f"; shows WORD_TO_REAL(CronEd.PR.Setpoint[50])/10; runs INTERN ASSIGN CronEd.PR.Setpoint[50]:=(REAL_TO_WORD(CronEd.PR_TT*10))
rounded rectangle at (420,290)-(451,311): text "%.1f"; shows WORD_TO_REAL(CronEd.PR.Setpoint[51])/10; runs INTERN ASSIGN CronEd.PR.Setpoint[51]:=(REAL_TO_WORD(CronEd.PR_TT*10))
rectangle at (420,200)-(451,221): text "h12"; runs INTERN ASSIGN CronEd.PR.Setpoint[51]:=(REAL_TO_WORD(CronEd.PR_TT*10));INTERN ASSIGN CronEd.PR.Setpoint[50]:=(REAL_TO_WORD(CronEd.PR_TT*10));INTERN ASSIGN CronEd.PR.Setpoint[49]:=(REAL_TO_WORD(CronEd.PR_TT*10));INTERN ASSIGN CronEd.PR.Setpoint[48]:=(REAL_TO_WORD(CronEd.PR_TT*10))
rounded rectangle at (450,230)-(481,251): text "%.1f"; shows WORD_TO_REAL(CronEd.PR.Setpoint[52])/10; runs INTERN ASSIGN CronEd.PR.Setpoint[52]:=(REAL_TO_WORD(CronEd.PR_TT*10))
rounded rectangle at (450,250)-(481,271): text "%.1f"; shows WORD_TO_REAL(CronEd.PR.Setpoint[53])/10; runs INTERN ASSIGN CronEd.PR.Setpoint[53]:=(REAL_TO_WORD(CronEd.PR_TT*10))
rounded rectangle at (450,270)-(481,291): text "%.1f"; shows WORD_TO_REAL(CronEd.PR.Setpoint[54])/10; runs INTERN ASSIGN CronEd.PR.Setpoint[54]:=(REAL_TO_WORD(CronEd.PR_TT*10))
rounded rectangle at (450,290)-(481,311): text "%.1f"; shows WORD_TO_REAL(CronEd.PR.Setpoint[55])/10; runs INTERN ASSIGN CronEd.PR.Setpoint[55]:=(REAL_TO_WORD(CronEd.PR_TT*10))
rectangle at (450,200)-(481,221): text "h13"; runs INTERN ASSIGN CronEd.PR.Setpoint[55]:=(REAL_TO_WORD(CronEd.PR_TT*10));INTERN ASSIGN CronEd.PR.Setpoint[54]:=(REAL_TO_WORD(CronEd.PR_TT*10));INTERN ASSIGN CronEd.PR.Setpoint[53]:=(REAL_TO_WORD(CronEd.PR_TT*10));INTERN ASSIGN CronEd.PR.Setpoint[52]:=(REAL_TO_WORD(CronEd.PR_TT*10))
rounded rectangle at (480,230)-(511,251): text "%.1f"; shows WORD_TO_REAL(CronEd.PR.Setpoint[56])/10; runs INTERN ASSIGN CronEd.PR.Setpoint[56]:=(REAL_TO_WORD(CronEd.PR_TT*10))
rounded rectangle at (480,250)-(511,271): text "%.1f"; shows WORD_TO_REAL(CronEd.PR.Setpoint[57])/10; runs INTERN ASSIGN CronEd.PR.Setpoint[57]:=(REAL_TO_WORD(CronEd.PR_TT*10))
rounded rectangle at (480,270)-(511,291): text "%.1f"; shows WORD_TO_REAL(CronEd.PR.Setpoint[58])/10; runs INTERN ASSIGN CronEd.PR.Setpoint[58]:=(REAL_TO_WORD(CronEd.PR_TT*10))
rounded rectangle at (480,290)-(511,311): text "%.1f"; shows WORD_TO_REAL(CronEd.PR.Setpoint[59])/10; runs INTERN ASSIGN CronEd.PR.Setpoint[59]:=(REAL_TO_WORD(CronEd.PR_TT*10))
rectangle at (480,200)-(511,221): text "h14"; runs INTERN ASSIGN CronEd.PR.Setpoint[59]:=(REAL_TO_WORD(CronEd.PR_TT*10));INTERN ASSIGN CronEd.PR.Setpoint[58]:=(REAL_TO_WORD(CronEd.PR_TT*10));INTERN ASSIGN CronEd.PR.Setpoint[57]:=(REAL_TO_WORD(CronEd.PR_TT*10));INTERN ASSIGN CronEd.PR.Setpoint[56]:=(REAL_TO_WORD(CronEd.PR_TT*10))
rounded rectangle at (510,230)-(541,251): text "%.1f"; shows WORD_TO_REAL(CronEd.PR.Setpoint[60])/10; runs INTERN ASSIGN CronEd.PR.Setpoint[60]:=(REAL_TO_WORD(CronEd.PR_TT*10))
rounded rectangle at (510,250)-(541,271): text "%.1f"; shows WORD_TO_REAL(CronEd.PR.Setpoint[61])/10; runs INTERN ASSIGN CronEd.PR.Setpoint[61]:=(REAL_TO_WORD(CronEd.PR_TT*10))
rounded rectangle at (510,270)-(541,291): text "%.1f"; shows WORD_TO_REAL(CronEd.PR.Setpoint[62])/10; runs INTERN ASSIGN CronEd.PR.Setpoint[62]:=(REAL_TO_WORD(CronEd.PR_TT*10))
rounded rectangle at (510,290)-(541,311): text "%.1f"; shows WORD_TO_REAL(CronEd.PR.Setpoint[63])/10; runs INTERN ASSIGN CronEd.PR.Setpoint[63]:=(REAL_TO_WORD(CronEd.PR_TT*10))
rectangle at (510,200)-(541,221): text "h15"; runs INTERN ASSIGN CronEd.PR.Setpoint[63]:=(REAL_TO_WORD(CronEd.PR_TT*10));INTERN ASSIGN CronEd.PR.Setpoint[62]:=(REAL_TO_WORD(CronEd.PR_TT*10));INTERN ASSIGN CronEd.PR.Setpoint[61]:=(REAL_TO_WORD(CronEd.PR_TT*10));INTERN ASSIGN CronEd.PR.Setpoint[60]:=(REAL_TO_WORD(CronEd.PR_TT*10))
rounded rectangle at (540,230)-(571,251): text "%.1f"; shows WORD_TO_REAL(CronEd.PR.Setpoint[64])/10; runs INTERN ASSIGN CronEd.PR.Setpoint[64]:=(REAL_TO_WORD(CronEd.PR_TT*10))
rounded rectangle at (540,250)-(571,271): text "%.1f"; shows WORD_TO_REAL(CronEd.PR.Setpoint[65])/10; runs INTERN ASSIGN CronEd.PR.Setpoint[65]:=(REAL_TO_WORD(CronEd.PR_TT*10))
rounded rectangle at (540,270)-(571,291): text "%.1f"; shows WORD_TO_REAL(CronEd.PR.Setpoint[66])/10; runs INTERN ASSIGN CronEd.PR.Setpoint[66]:=(REAL_TO_WORD(CronEd.PR_TT*10))
rounded rectangle at (540,290)-(571,311): text "%.1f"; shows WORD_TO_REAL(CronEd.PR.Setpoint[67])/10; runs INTERN ASSIGN CronEd.PR.Setpoint[67]:=(REAL_TO_WORD(CronEd.PR_TT*10))
rectangle at (540,200)-(571,221): text "h16"; runs INTERN ASSIGN CronEd.PR.Setpoint[67]:=(REAL_TO_WORD(CronEd.PR_TT*10));INTERN ASSIGN CronEd.PR.Setpoint[66]:=(REAL_TO_WORD(CronEd.PR_TT*10));INTERN ASSIGN CronEd.PR.Setpoint[65]:=(REAL_TO_WORD(CronEd.PR_TT*10));INTERN ASSIGN CronEd.PR.Setpoint[64]:=(REAL_TO_WORD(CronEd.PR_TT*10))
rounded rectangle at (570,230)-(601,251): text "%.1f"; shows WORD_TO_REAL(CronEd.PR.Setpoint[68])/10; runs INTERN ASSIGN CronEd.PR.Setpoint[68]:=(REAL_TO_WORD(CronEd.PR_TT*10))
rounded rectangle at (570,250)-(601,271): text "%.1f"; shows WORD_TO_REAL(CronEd.PR.Setpoint[69])/10; runs INTERN ASSIGN CronEd.PR.Setpoint[69]:=(REAL_TO_WORD(CronEd.PR_TT*10))
rounded rectangle at (570,270)-(601,291): text "%.1f"; shows WORD_TO_REAL(CronEd.PR.Setpoint[70])/10; runs INTERN ASSIGN CronEd.PR.Setpoint[70]:=(REAL_TO_WORD(CronEd.PR_TT*10))
rounded rectangle at (570,290)-(601,311): text "%.1f"; shows WORD_TO_REAL(CronEd.PR.Setpoint[71])/10; runs INTERN ASSIGN CronEd.PR.Setpoint[71]:=(REAL_TO_WORD(CronEd.PR_TT*10))
rectangle at (570,200)-(601,221): text "h17"; runs INTERN ASSIGN CronEd.PR.Setpoint[71]:=(REAL_TO_WORD(CronEd.PR_TT*10));INTERN ASSIGN CronEd.PR.Setpoint[70]:=(REAL_TO_WORD(CronEd.PR_TT*10));INTERN ASSIGN CronEd.PR.Setpoint[69]:=(REAL_TO_WORD(CronEd.PR_TT*10));INTERN ASSIGN CronEd.PR.Setpoint[68]:=(REAL_TO_WORD(CronEd.PR_TT*10))
rounded rectangle at (600,230)-(631,251): text "%.1f"; shows WORD_TO_REAL(CronEd.PR.Setpoint[72])/10; runs INTERN ASSIGN CronEd.PR.Setpoint[72]:=(REAL_TO_WORD(CronEd.PR_TT*10))
rounded rectangle at (600,250)-(631,271): text "%.1f"; shows WORD_TO_REAL(CronEd.PR.Setpoint[73])/10; runs INTERN ASSIGN CronEd.PR.Setpoint[73]:=(REAL_TO_WORD(CronEd.PR_TT*10))
rounded rectangle at (600,270)-(631,291): text "%.1f"; shows WORD_TO_REAL(CronEd.PR.Setpoint[74])/10; runs INTERN ASSIGN CronEd.PR.Setpoint[74]:=(REAL_TO_WORD(CronEd.PR_TT*10))
rounded rectangle at (600,290)-(631,311): text "%.1f"; shows WORD_TO_REAL(CronEd.PR.Setpoint[75])/10; runs INTERN ASSIGN CronEd.PR.Setpoint[75]:=(REAL_TO_WORD(CronEd.PR_TT*10))
rectangle at (600,200)-(631,221): text "h18"; runs INTERN ASSIGN CronEd.PR.Setpoint[75]:=(REAL_TO_WORD(CronEd.PR_TT*10));INTERN ASSIGN CronEd.PR.Setpoint[74]:=(REAL_TO_WORD(CronEd.PR_TT*10));INTERN ASSIGN CronEd.PR.Setpoint[73]:=(REAL_TO_WORD(CronEd.PR_TT*10));INTERN ASSIGN CronEd.PR.Setpoint[72]:=(REAL_TO_WORD(CronEd.PR_TT*10))
rounded rectangle at (630,230)-(661,251): text "%.1f"; shows WORD_TO_REAL(CronEd.PR.Setpoint[76])/10; runs INTERN ASSIGN CronEd.PR.Setpoint[76]:=(REAL_TO_WORD(CronEd.PR_TT*10))
rounded rectangle at (630,250)-(661,271): text "%.1f"; shows WORD_TO_REAL(CronEd.PR.Setpoint[77])/10; runs INTERN ASSIGN CronEd.PR.Setpoint[77]:=(REAL_TO_WORD(CronEd.PR_TT*10))
rounded rectangle at (630,270)-(661,291): text "%.1f"; shows WORD_TO_REAL(CronEd.PR.Setpoint[78])/10; runs INTERN ASSIGN CronEd.PR.Setpoint[78]:=(REAL_TO_WORD(CronEd.PR_TT*10))
rounded rectangle at (630,290)-(661,311): text "%.1f"; shows WORD_TO_REAL(CronEd.PR.Setpoint[79])/10; runs INTERN ASSIGN CronEd.PR.Setpoint[79]:=(REAL_TO_WORD(CronEd.PR_TT*10))
rectangle at (630,200)-(661,221): text "h19"; runs INTERN ASSIGN CronEd.PR.Setpoint[79]:=(REAL_TO_WORD(CronEd.PR_TT*10));INTERN ASSIGN CronEd.PR.Setpoint[78]:=(REAL_TO_WORD(CronEd.PR_TT*10));INTERN ASSIGN CronEd.PR.Setpoint[77]:=(REAL_TO_WORD(CronEd.PR_TT*10));INTERN ASSIGN CronEd.PR.Setpoint[76]:=(REAL_TO_WORD(CronEd.PR_TT*10))
rounded rectangle at (660,230)-(691,251): text "%.1f"; shows WORD_TO_REAL(CronEd.PR.Setpoint[80])/10; runs INTERN ASSIGN CronEd.PR.Setpoint[80]:=(REAL_TO_WORD(CronEd.PR_TT*10))
rounded rectangle at (660,250)-(691,271): text "%.1f"; shows WORD_TO_REAL(CronEd.PR.Setpoint[81])/10; runs INTERN ASSIGN CronEd.PR.Setpoint[81]:=(REAL_TO_WORD(CronEd.PR_TT*10))
rounded rectangle at (660,270)-(691,291): text "%.1f"; shows WORD_TO_REAL(CronEd.PR.Setpoint[82])/10; runs INTERN ASSIGN CronEd.PR.Setpoint[82]:=(REAL_TO_WORD(CronEd.PR_TT*10))
rounded rectangle at (660,290)-(691,311): text "%.1f"; shows WORD_TO_REAL(CronEd.PR.Setpoint[83])/10; runs INTERN ASSIGN CronEd.PR.Setpoint[83]:=(REAL_TO_WORD(CronEd.PR_TT*10))
rectangle at (660,200)-(691,221): text "h20"; runs INTERN ASSIGN CronEd.PR.Setpoint[83]:=(REAL_TO_WORD(CronEd.PR_TT*10));INTERN ASSIGN CronEd.PR.Setpoint[82]:=(REAL_TO_WORD(CronEd.PR_TT*10));INTERN ASSIGN CronEd.PR.Setpoint[81]:=(REAL_TO_WORD(CronEd.PR_TT*10));INTERN ASSIGN CronEd.PR.Setpoint[80]:=(REAL_TO_WORD(CronEd.PR_TT*10))
rounded rectangle at (690,230)-(721,251): text "%.1f"; shows WORD_TO_REAL(CronEd.PR.Setpoint[84])/10; runs INTERN ASSIGN CronEd.PR.Setpoint[84]:=(REAL_TO_WORD(CronEd.PR_TT*10))
rounded rectangle at (690,250)-(721,271): text "%.1f"; shows WORD_TO_REAL(CronEd.PR.Setpoint[85])/10; runs INTERN ASSIGN CronEd.PR.Setpoint[85]:=(REAL_TO_WORD(CronEd.PR_TT*10))
rounded rectangle at (690,270)-(721,291): text "%.1f"; shows WORD_TO_REAL(CronEd.PR.Setpoint[86])/10; runs INTERN ASSIGN CronEd.PR.Setpoint[86]:=(REAL_TO_WORD(CronEd.PR_TT*10))
rounded rectangle at (690,290)-(721,311): text "%.1f"; shows WORD_TO_REAL(CronEd.PR.Setpoint[87])/10; runs INTERN ASSIGN CronEd.PR.Setpoint[87]:=(REAL_TO_WORD(CronEd.PR_TT*10))
rectangle at (690,200)-(721,221): text "h21"; runs INTERN ASSIGN CronEd.PR.Setpoint[87]:=(REAL_TO_WORD(CronEd.PR_TT*10));INTERN ASSIGN CronEd.PR.Setpoint[86]:=(REAL_TO_WORD(CronEd.PR_TT*10));INTERN ASSIGN CronEd.PR.Setpoint[85]:=(REAL_TO_WORD(CronEd.PR_TT*10));INTERN ASSIGN CronEd.PR.Setpoint[84]:=(REAL_TO_WORD(CronEd.PR_TT*10))
rounded rectangle at (720,230)-(751,251): text "%.1f"; shows WORD_TO_REAL(CronEd.PR.Setpoint[88])/10; runs INTERN ASSIGN CronEd.PR.Setpoint[88]:=(REAL_TO_WORD(CronEd.PR_TT*10))
rounded rectangle at (720,250)-(751,271): text "%.1f"; shows WORD_TO_REAL(CronEd.PR.Setpoint[89])/10; runs INTERN ASSIGN CronEd.PR.Setpoint[89]:=(REAL_TO_WORD(CronEd.PR_TT*10))
rounded rectangle at (720,270)-(751,291): text "%.1f"; shows WORD_TO_REAL(CronEd.PR.Setpoint[90])/10; runs INTERN ASSIGN CronEd.PR.Setpoint[90]:=(REAL_TO_WORD(CronEd.PR_TT*10))
rounded rectangle at (720,290)-(751,311): text "%.1f"; shows WORD_TO_REAL(CronEd.PR.Setpoint[91])/10; runs INTERN ASSIGN CronEd.PR.Setpoint[91]:=(REAL_TO_WORD(CronEd.PR_TT*10))
rectangle at (720,200)-(751,221): text "h22"; runs INTERN ASSIGN CronEd.PR.Setpoint[91]:=(REAL_TO_WORD(CronEd.PR_TT*10));INTERN ASSIGN CronEd.PR.Setpoint[90]:=(REAL_TO_WORD(CronEd.PR_TT*10));INTERN ASSIGN CronEd.PR.Setpoint[89]:=(REAL_TO_WORD(CronEd.PR_TT*10));INTERN ASSIGN CronEd.PR.Setpoint[88]:=(REAL_TO_WORD(CronEd.PR_TT*10))
rounded rectangle at (750,230)-(781,251): text "%.1f"; shows WORD_TO_REAL(CronEd.PR.Setpoint[92])/10; runs INTERN ASSIGN CronEd.PR.Setpoint[92]:=(REAL_TO_WORD(CronEd.PR_TT*10))
rounded rectangle at (750,250)-(781,271): text "%.1f"; shows WORD_TO_REAL(CronEd.PR.Setpoint[93])/10; runs INTERN ASSIGN CronEd.PR.Setpoint[93]:=(REAL_TO_WORD(CronEd.PR_TT*10))
rounded rectangle at (750,270)-(781,291): text "%.1f"; shows WORD_TO_REAL(CronEd.PR.Setpoint[94])/10; runs INTERN ASSIGN CronEd.PR.Setpoint[94]:=(REAL_TO_WORD(CronEd.PR_TT*10))
rounded rectangle at (750,290)-(781,311): text "%.1f"; shows WORD_TO_REAL(CronEd.PR.Setpoint[95])/10; runs INTERN ASSIGN CronEd.PR.Setpoint[95]:=(REAL_TO_WORD(CronEd.PR_TT*10))
rectangle at (750,200)-(781,221): text "h23"; runs INTERN ASSIGN CronEd.PR.Setpoint[95]:=(REAL_TO_WORD(CronEd.PR_TT*10));INTERN ASSIGN CronEd.PR.Setpoint[94]:=(REAL_TO_WORD(CronEd.PR_TT*10));INTERN ASSIGN CronEd.PR.Setpoint[93]:=(REAL_TO_WORD(CronEd.PR_TT*10));INTERN ASSIGN CronEd.PR.Setpoint[92]:=(REAL_TO_WORD(CronEd.PR_TT*10))
rectangle at (410,360)-(491,381): text "Month"
rectangle at (490,360)-(531,381): text "%d"; shows CronEd.CA_Sel; alarm colour if CronEd.CA_Sel<>CronEd.CA_Act; editable 1..12
rectangle at (410,390)-(491,411): text "Profile Nr."
rectangle at (490,390)-(531,411): text "%d"; shows CronEd.CA_TPR; editable 0..10
button at (540,360)-(601,381): text "Load"; toggles CronEd.CA_Load
button at (610,360)-(671,381): text "Save"; toggles CronEd.CA_Save
rounded rectangle at (160,360)-(191,381): text "%d"; shows CronEd.CA.Profile[0]; invisible if CronEd.CA_DayF>0; alarm colour if CronEd.CA.Profile[0]=0; runs INTERN ASSIGN CronEd.CA.Profile[0]:=(CronEd.CA_TPR)
rectangle at (120,360)-(151,381): text "1"
rounded rectangle at (190,360)-(221,381): text "%d"; shows CronEd.CA.Profile[1]; invisible if CronEd.CA_DayF>1; alarm colour if CronEd.CA.Profile[1]=0; runs INTERN ASSIGN CronEd.CA.Profile[1]:=(CronEd.CA_TPR)
rounded rectangle at (220,360)-(251,381): text "%d"; shows CronEd.CA.Profile[2]; invisible if CronEd.CA_DayF>2; alarm colour if CronEd.CA.Profile[2]=0; runs INTERN ASSIGN CronEd.CA.Profile[2]:=(CronEd.CA_TPR)
rounded rectangle at (250,360)-(281,381): text "%d"; shows CronEd.CA.Profile[3]; invisible if CronEd.CA_DayF>3; alarm colour if CronEd.CA.Profile[3]=0; runs INTERN ASSIGN CronEd.CA.Profile[3]:=(CronEd.CA_TPR)
rounded rectangle at (280,360)-(311,381): text "%d"; shows CronEd.CA.Profile[4]; invisible if CronEd.CA_DayF>4; alarm colour if CronEd.CA.Profile[4]=0; runs INTERN ASSIGN CronEd.CA.Profile[4]:=(CronEd.CA_TPR)
rounded rectangle at (310,360)-(341,381): text "%d"; shows CronEd.CA.Profile[5]; invisible if CronEd.CA_DayF>5; alarm colour if CronEd.CA.Profile[5]=0; runs INTERN ASSIGN CronEd.CA.Profile[5]:=(CronEd.CA_TPR)
rounded rectangle at (340,360)-(371,381): text "%d"; shows CronEd.CA.Profile[6]; alarm colour if CronEd.CA.Profile[6]=0; runs INTERN ASSIGN CronEd.CA.Profile[6]:=(CronEd.CA_TPR)
rounded rectangle at (160,380)-(191,401): text "%d"; shows CronEd.CA.Profile[7]; alarm colour if CronEd.CA.Profile[7]=0; runs INTERN ASSIGN CronEd.CA.Profile[7]:=(CronEd.CA_TPR)
rectangle at (120,380)-(151,401): text "8"
rounded rectangle at (190,380)-(221,401): text "%d"; shows CronEd.CA.Profile[8]; alarm colour if CronEd.CA.Profile[8]=0; runs INTERN ASSIGN CronEd.CA.Profile[8]:=(CronEd.CA_TPR)
rounded rectangle at (220,380)-(251,401): text "%d"; shows CronEd.CA.Profile[9]; alarm colour if CronEd.CA.Profile[9]=0; runs INTERN ASSIGN CronEd.CA.Profile[9]:=(CronEd.CA_TPR)
rounded rectangle at (250,380)-(281,401): text "%d"; shows CronEd.CA.Profile[10]; alarm colour if CronEd.CA.Profile[10]=0; runs INTERN ASSIGN CronEd.CA.Profile[10]:=(CronEd.CA_TPR)
rounded rectangle at (280,380)-(311,401): text "%d"; shows CronEd.CA.Profile[11]; alarm colour if CronEd.CA.Profile[11]=0; runs INTERN ASSIGN CronEd.CA.Profile[11]:=(CronEd.CA_TPR)
rounded rectangle at (310,380)-(341,401): text "%d"; shows CronEd.CA.Profile[12]; alarm colour if CronEd.CA.Profile[12]=0; runs INTERN ASSIGN CronEd.CA.Profile[12]:=(CronEd.CA_TPR)
rounded rectangle at (340,380)-(371,401): text "%d"; shows CronEd.CA.Profile[13]; alarm colour if CronEd.CA.Profile[13]=0; runs INTERN ASSIGN CronEd.CA.Profile[13]:=(CronEd.CA_TPR)
rounded rectangle at (160,400)-(191,421): text "%d"; shows CronEd.CA.Profile[14]; alarm colour if CronEd.CA.Profile[14]=0; runs INTERN ASSIGN CronEd.CA.Profile[14]:=(CronEd.CA_TPR)
rectangle at (120,400)-(151,421): text "15"
rounded rectangle at (190,400)-(221,421): text "%d"; shows CronEd.CA.Profile[15]; alarm colour if CronEd.CA.Profile[15]=0; runs INTERN ASSIGN CronEd.CA.Profile[15]:=(CronEd.CA_TPR)
rounded rectangle at (220,400)-(251,421): text "%d"; shows CronEd.CA.Profile[16]; alarm colour if CronEd.CA.Profile[16]=0; runs INTERN ASSIGN CronEd.CA.Profile[16]:=(CronEd.CA_TPR)
rounded rectangle at (250,400)-(281,421): text "%d"; shows CronEd.CA.Profile[17]; alarm colour if CronEd.CA.Profile[17]=0; runs INTERN ASSIGN CronEd.CA.Profile[17]:=(CronEd.CA_TPR)
rounded rectangle at (280,400)-(311,421): text "%d"; shows CronEd.CA.Profile[18]; alarm colour if CronEd.CA.Profile[18]=0; runs INTERN ASSIGN CronEd.CA.Profile[18]:=(CronEd.CA_TPR)
rounded rectangle at (310,400)-(341,421): text "%d"; shows CronEd.CA.Profile[19]; alarm colour if CronEd.CA.Profile[19]=0; runs INTERN ASSIGN CronEd.CA.Profile[19]:=(CronEd.CA_TPR)
rounded rectangle at (340,400)-(371,421): text "%d"; shows CronEd.CA.Profile[20]; alarm colour if CronEd.CA.Profile[20]=0; runs INTERN ASSIGN CronEd.CA.Profile[20]:=(CronEd.CA_TPR)
rounded rectangle at (160,420)-(191,441): text "%d"; shows CronEd.CA.Profile[21]; alarm colour if CronEd.CA.Profile[21]=0; runs INTERN ASSIGN CronEd.CA.Profile[21]:=(CronEd.CA_TPR)
rectangle at (120,420)-(151,441): text "22"
rounded rectangle at (190,420)-(221,441): text "%d"; shows CronEd.CA.Profile[22]; alarm colour if CronEd.CA.Profile[22]=0; runs INTERN ASSIGN CronEd.CA.Profile[22]:=(CronEd.CA_TPR)
rounded rectangle at (220,420)-(251,441): text "%d"; shows CronEd.CA.Profile[23]; alarm colour if CronEd.CA.Profile[23]=0; runs INTERN ASSIGN CronEd.CA.Profile[23]:=(CronEd.CA_TPR)
rounded rectangle at (250,420)-(281,441): text "%d"; shows CronEd.CA.Profile[24]; alarm colour if CronEd.CA.Profile[24]=0; runs INTERN ASSIGN CronEd.CA.Profile[24]:=(CronEd.CA_TPR)
rounded rectangle at (280,420)-(311,441): text "%d"; shows CronEd.CA.Profile[25]; alarm colour if CronEd.CA.Profile[25]=0; runs INTERN ASSIGN CronEd.CA.Profile[25]:=(CronEd.CA_TPR)
rounded rectangle at (310,420)-(341,441): text "%d"; shows CronEd.CA.Profile[26]; alarm colour if CronEd.CA.Profile[26]=0; runs INTERN ASSIGN CronEd.CA.Profile[26]:=(CronEd.CA_TPR)
rounded rectangle at (340,420)-(371,441): text "%d"; shows CronEd.CA.Profile[27]; alarm colour if CronEd.CA.Profile[27]=0; runs INTERN ASSIGN CronEd.CA.Profile[27]:=(CronEd.CA_TPR)
rounded rectangle at (160,440)-(191,461): text "%d"; shows CronEd.CA.Profile[28]; alarm colour if CronEd.CA.Profile[28]=0; runs INTERN ASSIGN CronEd.CA.Profile[28]:=(CronEd.CA_TPR)
rectangle at (120,440)-(151,461): text "29"
rounded rectangle at (190,440)-(221,461): text "%d"; shows CronEd.CA.Profile[29]; alarm colour if CronEd.CA.Profile[29]=0; runs INTERN ASSIGN CronEd.CA.Profile[29]:=(CronEd.CA_TPR)
rounded rectangle at (220,440)-(251,461): text "%d"; shows CronEd.CA.Profile[30]; alarm colour if CronEd.CA.Profile[30]=0; runs INTERN ASSIGN CronEd.CA.Profile[30]:=(CronEd.CA_TPR)
rounded rectangle at (250,440)-(281,461): text "%d"; shows CronEd.CA.Profile[31]; alarm colour if CronEd.CA.Profile[31]=0; runs INTERN ASSIGN CronEd.CA.Profile[31]:=(CronEd.CA_TPR)
rounded rectangle at (280,440)-(311,461): text "%d"; shows CronEd.CA.Profile[32]; invisible if CronEd.CA_DayL<32; alarm colour if CronEd.CA.Profile[32]=0; runs INTERN ASSIGN CronEd.CA.Profile[32]:=(CronEd.CA_TPR)
rounded rectangle at (310,440)-(341,461): text "%d"; shows CronEd.CA.Profile[33]; invisible if CronEd.CA_DayL<33; alarm colour if CronEd.CA.Profile[33]=0; runs INTERN ASSIGN CronEd.CA.Profile[33]:=(CronEd.CA_TPR)
rounded rectangle at (340,440)-(371,461): text "%d"; shows CronEd.CA.Profile[34]; invisible if CronEd.CA_DayL<34; alarm colour if CronEd.CA.Profile[34]=0; runs INTERN ASSIGN CronEd.CA.Profile[34]:=(CronEd.CA_TPR)
rounded rectangle at (160,460)-(191,481): text "%d"; shows CronEd.CA.Profile[35]; invisible if CronEd.CA_DayL<35; alarm colour if CronEd.CA.Profile[35]=0; runs INTERN ASSIGN CronEd.CA.Profile[35]:=(CronEd.CA_TPR)
rectangle at (120,460)-(151,481): text "36"; invisible if CronEd.CA_DayL<35
rounded rectangle at (190,460)-(221,481): text "%d"; shows CronEd.CA.Profile[36]; invisible if CronEd.CA_DayL<36; alarm colour if CronEd.CA.Profile[36]=0; runs INTERN ASSIGN CronEd.CA.Profile[36]:=(CronEd.CA_TPR)
rounded rectangle at (220,460)-(251,481): text "%d"; shows CronEd.CA.Profile[37]; invisible if CronEd.CA_DayL<37; alarm colour if CronEd.CA.Profile[37]=0; runs INTERN ASSIGN CronEd.CA.Profile[37]:=(CronEd.CA_TPR)
rounded rectangle at (250,460)-(281,481): text "%d"; shows CronEd.CA.Profile[38]; invisible if CronEd.CA_DayL<38; alarm colour if CronEd.CA.Profile[38]=0; runs INTERN ASSIGN CronEd.CA.Profile[38]:=(CronEd.CA_TPR)
rounded rectangle at (280,460)-(311,481): text "%d"; shows CronEd.CA.Profile[39]; invisible if CronEd.CA_DayL<39; alarm colour if CronEd.CA.Profile[39]=0; runs INTERN ASSIGN CronEd.CA.Profile[39]:=(CronEd.CA_TPR)
rounded rectangle at (310,460)-(341,481): text "%d"; shows CronEd.CA.Profile[40]; invisible if CronEd.CA_DayL<40; alarm colour if CronEd.CA.Profile[40]=0; runs INTERN ASSIGN CronEd.CA.Profile[40]:=(CronEd.CA_TPR)
rounded rectangle at (340,460)-(371,481): text "%d"; shows CronEd.CA.Profile[41]; invisible if CronEd.CA_DayL<41; alarm colour if CronEd.CA.Profile[41]=0; runs INTERN ASSIGN CronEd.CA.Profile[41]:=(CronEd.CA_TPR)
rectangle at (310,60)-(371,81): text "Year"
rectangle at (370,60)-(411,81): text "%d"; shows CronEd.CN_YSel; alarm colour if CronEd.CN_YSel<>CronEd.CN_YAct; editable 2000..2100
rectangle at (480,60)-(761,81): text "%s"; shows CronEd.Message
button at (10,50)-(71,81): text "REINIT"; runs INTERN ASSIGN THER01.InitOK:=(FALSE);INTERN ASSIGN THER02.InitOK:=(FALSE);INTERN ASSIGN THER03.InitOK:=(FALSE);INTERN ASSIGN THER04.InitOK:=(FALSE);INTERN ASSIGN THER05.InitOK:=(FALSE)
2 more shapes without text or variables
*)

(* Visualisation VIS_SET
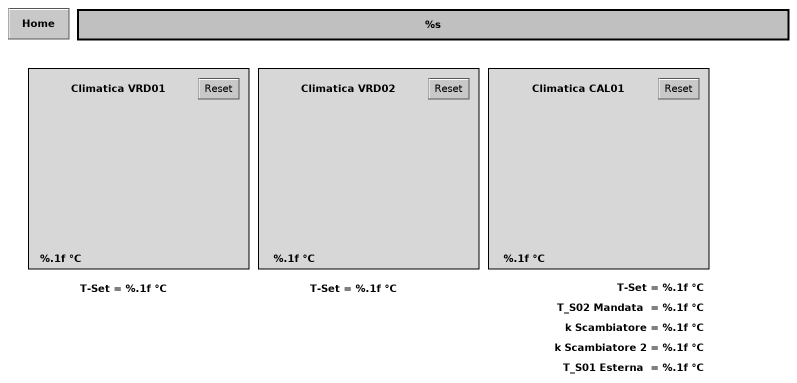
rectangle at (40,80)-(201,101): text "Climatica VRD01"
button at (200,80)-(241,101): text "Reset"; taps .VRD01.CLIM.InitOK
button at (10,10)-(71,41): text "Home"; opens PLC_VISU
rectangle at (80,280)-(221,301): text "T-Set = %.1f °C"; shows INT_TO_REAL(.VRD01.Ctrl_SetPoint)/10
rectangle at (270,80)-(431,101): text "Climatica VRD02"
button at (430,80)-(471,101): text "Reset"; taps .VRD02.CLIM.InitOK; runs INTERN ASSIGN VRD02_Clima.InitOK:=(FALSE)
rectangle at (310,280)-(451,301): text "T-Set = %.1f °C"; shows INT_TO_REAL(.VRD02.Ctrl_SetPoint)/10
rectangle at (40,250)-(91,271): text "%.1f °C"; shows INT_TO_REAL(.TPV05.IN)/10
rectangle at (270,250)-(321,271): text "%.1f °C"; shows INT_TO_REAL(.TPV06.IN)/10
rectangle at (500,80)-(661,101): text "Climatica CAL01"
button at (660,80)-(701,101): text "Reset"; taps .CAL01.CLIM.InitOK; runs INTERN ASSIGN VRD02_Clima.InitOK:=(FALSE)
rectangle at (500,250)-(551,271): text "%.1f °C"; shows INT_TO_REAL(.TPV06.IN)/10
rectangle at (79,11)-(791,42): text "%s"; shows .Plant_NAME
rectangle at (567,279)-(708,300): text "T-Set = %.1f °C"; shows INT_TO_REAL(.CAL01.SetPoint)/10
rectangle at (547,319)-(708,340): text "k Scambiatore = %.1f °C"; shows INT_TO_REAL(.OffsetSetPointManuale/10)
rectangle at (547,339)-(708,360): text "k Scambiatore 2 = %.1f °C"; shows INT_TO_REAL(.OffsetSetPointManuale2/10)
rectangle at (537,359)-(708,380): text "T_S01 Esterna  = %.1f °C"; shows INT_TO_REAL(.TPV01.IN)/10
rectangle at (547,299)-(708,320): text "T_S02 Mandata  = %.1f °C"; shows INT_TO_REAL(.TPV02.AVG)/10
3 more shapes without text or variables
44 elements of other kinds (tables, trends, ...) not read
*)
